//     PlcTask Outputs/GVL_iXlinker.EtherCAT_Master_EPPxxxx.Beckhoff_EPP2xxx.Beckhoff_EPP2xxxEK1122.A_0071_EPP2809_0021_0016.Channel_5.Output <-> Channel 5/Output
//     PlcTask Outputs/GVL_iXlinker.EtherCAT_Master_EPPxxxx.Beckhoff_EPP2xxx.Beckhoff_EPP2xxxEK1122.A_0071_EPP2809_0021_0016.Channel_6.Output <-> Channel 6/Output
//     PlcTask Outputs/GVL_iXlinker.EtherCAT_Master_EPPxxxx.Beckhoff_EPP2xxx.Beckhoff_EPP2xxxEK1122.A_0071_EPP2809_0021_0016.Channel_7.Output <-> Channel 7/Output
//     PlcTask Outputs/GVL_iXlinker.EtherCAT_Master_EPPxxxx.Beckhoff_EPP2xxx.Beckhoff_EPP2xxxEK1122.A_0071_EPP2809_0021_0016.Channel_8.Output <-> Channel 8/Output
//     PlcTask Outputs/GVL_iXlinker.EtherCAT_Master_EPPxxxx.Beckhoff_EPP2xxx.Beckhoff_EPP2xxxEK1122.A_0071_EPP2809_0021_0016.Channel_9.Output <-> Channel 9/Output
//     PlcTask Outputs/GVL_iXlinker.EtherCAT_Master_EPPxxxx.Beckhoff_EPP2xxx.Beckhoff_EPP2xxxEK1122.A_0071_EPP2809_0021_0016.Channel_10.Output <-> Channel 10/Output
//     PlcTask Outputs/GVL_iXlinker.EtherCAT_Master_EPPxxxx.Beckhoff_EPP2xxx.Beckhoff_EPP2xxxEK1122.A_0071_EPP2809_0021_0016.Channel_11.Output <-> Channel 11/Output
//     PlcTask Outputs/GVL_iXlinker.EtherCAT_Master_EPPxxxx.Beckhoff_EPP2xxx.Beckhoff_EPP2xxxEK1122.A_0071_EPP2809_0021_0016.Channel_12.Output <-> Channel 12/Output
//     PlcTask Outputs/GVL_iXlinker.EtherCAT_Master_EPPxxxx.Beckhoff_EPP2xxx.Beckhoff_EPP2xxxEK1122.A_0071_EPP2809_0021_0016.Channel_13.Output <-> Channel 13/Output
//     PlcTask Outputs/GVL_iXlinker.EtherCAT_Master_EPPxxxx.Beckhoff_EPP2xxx.Beckhoff_EPP2xxxEK1122.A_0071_EPP2809_0021_0016.Channel_14.Output <-> Channel 14/Output
//     PlcTask Outputs/GVL_iXlinker.EtherCAT_Master_EPPxxxx.Beckhoff_EPP2xxx.Beckhoff_EPP2xxxEK1122.A_0071_EPP2809_0021_0016.Channel_15.Output <-> Channel 15/Output
//     PlcTask Outputs/GVL_iXlinker.EtherCAT_Master_EPPxxxx.Beckhoff_EPP2xxx.Beckhoff_EPP2xxxEK1122.A_0071_EPP2809_0021_0016.Channel_16.Output <-> Channel 16/Output
//     PlcTask Inputs/GVL_iXlinker.EtherCAT_Master_EPPxxxx.Beckhoff_EPP2xxx.Beckhoff_EPP2xxxEK1122.A_0071_EPP2809_0021_0016.WcState.WcState <-> WcState/WcState
//     PlcTask Inputs/GVL_iXlinker.EtherCAT_Master_EPPxxxx.Beckhoff_EPP2xxx.Beckhoff_EPP2xxxEK1122.A_0071_EPP2809_0021_0016.InfoData.State <-> InfoData/State
//   PLC/PLC Instance <-> EtherCAT Master EPPxxxx/Beckhoff EPP2xxx/Beckhoff EPP2xxxEK1122/A_0072(EPP2809-0022-0016)
//     PlcTask Outputs/GVL_iXlinker.EtherCAT_Master_EPPxxxx.Beckhoff_EPP2xxx.Beckhoff_EPP2xxxEK1122.A_0072_EPP2809_0022_0016.Channel_1.Output <-> Channel 1/Output
//     PlcTask Outputs/GVL_iXlinker.EtherCAT_Master_EPPxxxx.Beckhoff_EPP2xxx.Beckhoff_EPP2xxxEK1122.A_0072_EPP2809_0022_0016.Channel_2.Output <-> Channel 2/Output
//     PlcTask Outputs/GVL_iXlinker.EtherCAT_Master_EPPxxxx.Beckhoff_EPP2xxx.Beckhoff_EPP2xxxEK1122.A_0072_EPP2809_0022_0016.Channel_3.Output <-> Channel 3/Output
//     PlcTask Outputs/GVL_iXlinker.EtherCAT_Master_EPPxxxx.Beckhoff_EPP2xxx.Beckhoff_EPP2xxxEK1122.A_0072_EPP2809_0022_0016.Channel_4.Output <-> Channel 4/Output
//     PlcTask Outputs/GVL_iXlinker.EtherCAT_Master_EPPxxxx.Beckhoff_EPP2xxx.Beckhoff_EPP2xxxEK1122.A_0072_EPP2809_0022_0016.Channel_5.Output <-> Channel 5/Output
//     PlcTask Outputs/GVL_iXlinker.EtherCAT_Master_EPPxxxx.Beckhoff_EPP2xxx.Beckhoff_EPP2xxxEK1122.A_0072_EPP2809_0022_0016.Channel_6.Output <-> Channel 6/Output
//     PlcTask Outputs/GVL_iXlinker.EtherCAT_Master_EPPxxxx.Beckhoff_EPP2xxx.Beckhoff_EPP2xxxEK1122.A_0072_EPP2809_0022_0016.Channel_7.Output <-> Channel 7/Output
//     PlcTask Outputs/GVL_iXlinker.EtherCAT_Master_EPPxxxx.Beckhoff_EPP2xxx.Beckhoff_EPP2xxxEK1122.A_0072_EPP2809_0022_0016.Channel_8.Output <-> Channel 8/Output
//     PlcTask Outputs/GVL_iXlinker.EtherCAT_Master_EPPxxxx.Beckhoff_EPP2xxx.Beckhoff_EPP2xxxEK1122.A_0072_EPP2809_0022_0016.Channel_9.Output <-> Channel 9/Output
//     PlcTask Outputs/GVL_iXlinker.EtherCAT_Master_EPPxxxx.Beckhoff_EPP2xxx.Beckhoff_EPP2xxxEK1122.A_0072_EPP2809_0022_0016.Channel_10.Output <-> Channel 10/Output
//     PlcTask Outputs/GVL_iXlinker.EtherCAT_Master_EPPxxxx.Beckhoff_EPP2xxx.Beckhoff_EPP2xxxEK1122.A_0072_EPP2809_0022_0016.Channel_11.Output <-> Channel 11/Output
//     PlcTask Outputs/GVL_iXlinker.EtherCAT_Master_EPPxxxx.Beckhoff_EPP2xxx.Beckhoff_EPP2xxxEK1122.A_0072_EPP2809_0022_0016.Channel_12.Output <-> Channel 12/Output
//     PlcTask Outputs/GVL_iXlinker.EtherCAT_Master_EPPxxxx.Beckhoff_EPP2xxx.Beckhoff_EPP2xxxEK1122.A_0072_EPP2809_0022_0016.Channel_13.Output <-> Channel 13/Output
//     PlcTask Outputs/GVL_iXlinker.EtherCAT_Master_EPPxxxx.Beckhoff_EPP2xxx.Beckhoff_EPP2xxxEK1122.A_0072_EPP2809_0022_0016.Channel_14.Output <-> Channel 14/Output
//     PlcTask Outputs/GVL_iXlinker.EtherCAT_Master_EPPxxxx.Beckhoff_EPP2xxx.Beckhoff_EPP2xxxEK1122.A_0072_EPP2809_0022_0016.Channel_15.Output <-> Channel 15/Output
//     PlcTask Outputs/GVL_iXlinker.EtherCAT_Master_EPPxxxx.Beckhoff_EPP2xxx.Beckhoff_EPP2xxxEK1122.A_0072_EPP2809_0022_0016.Channel_16.Output <-> Channel 16/Output
//     PlcTask Inputs/GVL_iXlinker.EtherCAT_Master_EPPxxxx.Beckhoff_EPP2xxx.Beckhoff_EPP2xxxEK1122.A_0072_EPP2809_0022_0016.WcState.WcState <-> WcState/WcState
//     PlcTask Inputs/GVL_iXlinker.EtherCAT_Master_EPPxxxx.Beckhoff_EPP2xxx.Beckhoff_EPP2xxxEK1122.A_0072_EPP2809_0022_0016.InfoData.State <-> InfoData/State
//   PLC/PLC Instance <-> EtherCAT Master EPPxxxx/Beckhoff EPP2xxx/Beckhoff EPP2xxxEK1122/A_0073(EPP2816-0004-0016)
//     PlcTask Inputs/GVL_iXlinker.EtherCAT_Master_EPPxxxx.Beckhoff_EPP2xxx.Beckhoff_EPP2xxxEK1122.A_0073_EPP2816_0004_0016.DIG_Diag_Inputs_Channel_1.Diag_Input[0] <-> DIG Diag Inputs Channel 1/Diag Input 1
//     PlcTask Inputs/GVL_iXlinker.EtherCAT_Master_EPPxxxx.Beckhoff_EPP2xxx.Beckhoff_EPP2xxxEK1122.A_0073_EPP2816_0004_0016.DIG_Diag_Inputs_Channel_1.Diag_Input[1] <-> DIG Diag Inputs Channel 1/Diag Input 2
//     PlcTask Inputs/GVL_iXlinker.EtherCAT_Master_EPPxxxx.Beckhoff_EPP2xxx.Beckhoff_EPP2xxxEK1122.A_0073_EPP2816_0004_0016.DIG_Diag_Inputs_Channel_1.Diag_Input[2] <-> DIG Diag Inputs Channel 1/Diag Input 3
//     PlcTask Inputs/GVL_iXlinker.EtherCAT_Master_EPPxxxx.Beckhoff_EPP2xxx.Beckhoff_EPP2xxxEK1122.A_0073_EPP2816_0004_0016.DIG_Diag_Inputs_Channel_1.Diag_Input[3] <-> DIG Diag Inputs Channel 1/Diag Input 4
//     PlcTask Inputs/GVL_iXlinker.EtherCAT_Master_EPPxxxx.Beckhoff_EPP2xxx.Beckhoff_EPP2xxxEK1122.A_0073_EPP2816_0004_0016.DIG_Diag_Inputs_Channel_1.Diag_Input[4] <-> DIG Diag Inputs Channel 1/Diag Input 5
//     PlcTask Inputs/GVL_iXlinker.EtherCAT_Master_EPPxxxx.Beckhoff_EPP2xxx.Beckhoff_EPP2xxxEK1122.A_0073_EPP2816_0004_0016.DIG_Diag_Inputs_Channel_1.Diag_Input[5] <-> DIG Diag Inputs Channel 1/Diag Input 6
//     PlcTask Inputs/GVL_iXlinker.EtherCAT_Master_EPPxxxx.Beckhoff_EPP2xxx.Beckhoff_EPP2xxxEK1122.A_0073_EPP2816_0004_0016.DIG_Diag_Inputs_Channel_1.Diag_Input[6] <-> DIG Diag Inputs Channel 1/Diag Input 7
//     PlcTask Inputs/GVL_iXlinker.EtherCAT_Master_EPPxxxx.Beckhoff_EPP2xxx.Beckhoff_EPP2xxxEK1122.A_0073_EPP2816_0004_0016.DIG_Diag_Inputs_Channel_1.Diag_Input[7] <-> DIG Diag Inputs Channel 1/Diag Input 8
//     PlcTask Inputs/GVL_iXlinker.EtherCAT_Master_EPPxxxx.Beckhoff_EPP2xxx.Beckhoff_EPP2xxxEK1122.A_0073_EPP2816_0004_0016.DIG_Diag_Inputs_Channel_2.Diag_Input[0] <-> DIG Diag Inputs Channel 2/Diag Input 1
//     PlcTask Inputs/GVL_iXlinker.EtherCAT_Master_EPPxxxx.Beckhoff_EPP2xxx.Beckhoff_EPP2xxxEK1122.A_0073_EPP2816_0004_0016.DIG_Diag_Inputs_Channel_2.Diag_Input[1] <-> DIG Diag Inputs Channel 2/Diag Input 2
//     PlcTask Inputs/GVL_iXlinker.EtherCAT_Master_EPPxxxx.Beckhoff_EPP2xxx.Beckhoff_EPP2xxxEK1122.A_0073_EPP2816_0004_0016.DIG_Diag_Inputs_Channel_2.Diag_Input[2] <-> DIG Diag Inputs Channel 2/Diag Input 3
//     PlcTask Inputs/GVL_iXlinker.EtherCAT_Master_EPPxxxx.Beckhoff_EPP2xxx.Beckhoff_EPP2xxxEK1122.A_0073_EPP2816_0004_0016.DIG_Diag_Inputs_Channel_2.Diag_Input[3] <-> DIG Diag Inputs Channel 2/Diag Input 4
//     PlcTask Inputs/GVL_iXlinker.EtherCAT_Master_EPPxxxx.Beckhoff_EPP2xxx.Beckhoff_EPP2xxxEK1122.A_0073_EPP2816_0004_0016.DIG_Diag_Inputs_Channel_2.Diag_Input[4] <-> DIG Diag Inputs Channel 2/Diag Input 5
//     PlcTask Inputs/GVL_iXlinker.EtherCAT_Master_EPPxxxx.Beckhoff_EPP2xxx.Beckhoff_EPP2xxxEK1122.A_0073_EPP2816_0004_0016.DIG_Diag_Inputs_Channel_2.Diag_Input[5] <-> DIG Diag Inputs Channel 2/Diag Input 6
//     PlcTask Inputs/GVL_iXlinker.EtherCAT_Master_EPPxxxx.Beckhoff_EPP2xxx.Beckhoff_EPP2xxxEK1122.A_0073_EPP2816_0004_0016.DIG_Diag_Inputs_Channel_2.Diag_Input[6] <-> DIG Diag Inputs Channel 2/Diag Input 7
//     PlcTask Inputs/GVL_iXlinker.EtherCAT_Master_EPPxxxx.Beckhoff_EPP2xxx.Beckhoff_EPP2xxxEK1122.A_0073_EPP2816_0004_0016.DIG_Diag_Inputs_Channel_2.Diag_Input[7] <-> DIG Diag Inputs Channel 2/Diag Input 8
//     PlcTask Inputs/GVL_iXlinker.EtherCAT_Master_EPPxxxx.Beckhoff_EPP2xxx.Beckhoff_EPP2xxxEK1122.A_0073_EPP2816_0004_0016.DIG_Inputs_Device.Safe_state_active <-> DIG Inputs Device/Safe state active
//     PlcTask Inputs/GVL_iXlinker.EtherCAT_Master_EPPxxxx.Beckhoff_EPP2xxx.Beckhoff_EPP2xxxEK1122.A_0073_EPP2816_0004_0016.DIG_Inputs_Device.Error_channel[0] <-> DIG Inputs Device/Error channel 1
//     PlcTask Inputs/GVL_iXlinker.EtherCAT_Master_EPPxxxx.Beckhoff_EPP2xxx.Beckhoff_EPP2xxxEK1122.A_0073_EPP2816_0004_0016.DIG_Inputs_Device.Error_channel[1] <-> DIG Inputs Device/Error channel 2
//     PlcTask Inputs/GVL_iXlinker.EtherCAT_Master_EPPxxxx.Beckhoff_EPP2xxx.Beckhoff_EPP2xxxEK1122.A_0073_EPP2816_0004_0016.DIG_Inputs_Device.Sync_error <-> DIG Inputs Device/Sync error
//     PlcTask Inputs/GVL_iXlinker.EtherCAT_Master_EPPxxxx.Beckhoff_EPP2xxx.Beckhoff_EPP2xxxEK1122.A_0073_EPP2816_0004_0016.DIG_Inputs_Device.TxPDO_Toggle <-> DIG Inputs Device/TxPDO Toggle
//     PlcTask Outputs/GVL_iXlinker.EtherCAT_Master_EPPxxxx.Beckhoff_EPP2xxx.Beckhoff_EPP2xxxEK1122.A_0073_EPP2816_0004_0016.DIG_Output_Channel_1.Output[0] <-> DIG Output Channel 1/Output 1
//     PlcTask Outputs/GVL_iXlinker.EtherCAT_Master_EPPxxxx.Beckhoff_EPP2xxx.Beckhoff_EPP2xxxEK1122.A_0073_EPP2816_0004_0016.DIG_Output_Channel_1.Output[1] <-> DIG Output Channel 1/Output 2
//     PlcTask Outputs/GVL_iXlinker.EtherCAT_Master_EPPxxxx.Beckhoff_EPP2xxx.Beckhoff_EPP2xxxEK1122.A_0073_EPP2816_0004_0016.DIG_Output_Channel_1.Output[2] <-> DIG Output Channel 1/Output 3
//     PlcTask Outputs/GVL_iXlinker.EtherCAT_Master_EPPxxxx.Beckhoff_EPP2xxx.Beckhoff_EPP2xxxEK1122.A_0073_EPP2816_0004_0016.DIG_Output_Channel_1.Output[3] <-> DIG Output Channel 1/Output 4
//     PlcTask Outputs/GVL_iXlinker.EtherCAT_Master_EPPxxxx.Beckhoff_EPP2xxx.Beckhoff_EPP2xxxEK1122.A_0073_EPP2816_0004_0016.DIG_Output_Channel_1.Output[4] <-> DIG Output Channel 1/Output 5
//     PlcTask Outputs/GVL_iXlinker.EtherCAT_Master_EPPxxxx.Beckhoff_EPP2xxx.Beckhoff_EPP2xxxEK1122.A_0073_EPP2816_0004_0016.DIG_Output_Channel_1.Output[5] <-> DIG Output Channel 1/Output 6
//     PlcTask Outputs/GVL_iXlinker.EtherCAT_Master_EPPxxxx.Beckhoff_EPP2xxx.Beckhoff_EPP2xxxEK1122.A_0073_EPP2816_0004_0016.DIG_Output_Channel_1.Output[6] <-> DIG Output Channel 1/Output 7
//     PlcTask Outputs/GVL_iXlinker.EtherCAT_Master_EPPxxxx.Beckhoff_EPP2xxx.Beckhoff_EPP2xxxEK1122.A_0073_EPP2816_0004_0016.DIG_Output_Channel_1.Output[7] <-> DIG Output Channel 1/Output 8
//     PlcTask Outputs/GVL_iXlinker.EtherCAT_Master_EPPxxxx.Beckhoff_EPP2xxx.Beckhoff_EPP2xxxEK1122.A_0073_EPP2816_0004_0016.DIG_Output_Channel_2.Output[0] <-> DIG Output Channel 2/Output 1
//     PlcTask Outputs/GVL_iXlinker.EtherCAT_Master_EPPxxxx.Beckhoff_EPP2xxx.Beckhoff_EPP2xxxEK1122.A_0073_EPP2816_0004_0016.DIG_Output_Channel_2.Output[1] <-> DIG Output Channel 2/Output 2
//     PlcTask Outputs/GVL_iXlinker.EtherCAT_Master_EPPxxxx.Beckhoff_EPP2xxx.Beckhoff_EPP2xxxEK1122.A_0073_EPP2816_0004_0016.DIG_Output_Channel_2.Output[2] <-> DIG Output Channel 2/Output 3
//     PlcTask Outputs/GVL_iXlinker.EtherCAT_Master_EPPxxxx.Beckhoff_EPP2xxx.Beckhoff_EPP2xxxEK1122.A_0073_EPP2816_0004_0016.DIG_Output_Channel_2.Output[3] <-> DIG Output Channel 2/Output 4
//     PlcTask Outputs/GVL_iXlinker.EtherCAT_Master_EPPxxxx.Beckhoff_EPP2xxx.Beckhoff_EPP2xxxEK1122.A_0073_EPP2816_0004_0016.DIG_Output_Channel_2.Output[4] <-> DIG Output Channel 2/Output 5
//     PlcTask Outputs/GVL_iXlinker.EtherCAT_Master_EPPxxxx.Beckhoff_EPP2xxx.Beckhoff_EPP2xxxEK1122.A_0073_EPP2816_0004_0016.DIG_Output_Channel_2.Output[5] <-> DIG Output Channel 2/Output 6
//     PlcTask Outputs/GVL_iXlinker.EtherCAT_Master_EPPxxxx.Beckhoff_EPP2xxx.Beckhoff_EPP2xxxEK1122.A_0073_EPP2816_0004_0016.DIG_Output_Channel_2.Output[6] <-> DIG Output Channel 2/Output 7
//     PlcTask Outputs/GVL_iXlinker.EtherCAT_Master_EPPxxxx.Beckhoff_EPP2xxx.Beckhoff_EPP2xxxEK1122.A_0073_EPP2816_0004_0016.DIG_Output_Channel_2.Output[7] <-> DIG Output Channel 2/Output 8
//     PlcTask Outputs/GVL_iXlinker.EtherCAT_Master_EPPxxxx.Beckhoff_EPP2xxx.Beckhoff_EPP2xxxEK1122.A_0073_EPP2816_0004_0016.DIG_Outputs_Device.Set_safe_state <-> DIG Outputs Device/Set safe state
//     PlcTask Outputs/GVL_iXlinker.EtherCAT_Master_EPPxxxx.Beckhoff_EPP2xxx.Beckhoff_EPP2xxxEK1122.A_0073_EPP2816_0004_0016.DIG_Outputs_Device.Reset_outputs <-> DIG Outputs Device/Reset outputs
//     PlcTask Inputs/GVL_iXlinker.EtherCAT_Master_EPPxxxx.Beckhoff_EPP2xxx.Beckhoff_EPP2xxxEK1122.A_0073_EPP2816_0004_0016.WcState.WcState <-> WcState/WcState
//     PlcTask Inputs/GVL_iXlinker.EtherCAT_Master_EPPxxxx.Beckhoff_EPP2xxx.Beckhoff_EPP2xxxEK1122.A_0073_EPP2816_0004_0016.WcState.InputToggle <-> WcState/InputToggle
//     PlcTask Inputs/GVL_iXlinker.EtherCAT_Master_EPPxxxx.Beckhoff_EPP2xxx.Beckhoff_EPP2xxxEK1122.A_0073_EPP2816_0004_0016.InfoData.AdsAddr <-> InfoData/AdsAddr
//     PlcTask Inputs/GVL_iXlinker.EtherCAT_Master_EPPxxxx.Beckhoff_EPP2xxx.Beckhoff_EPP2xxxEK1122.A_0073_EPP2816_0004_0016.InfoData.State <-> InfoData/State
//   PLC/PLC Instance <-> EtherCAT Master EPPxxxx/Beckhoff EPP2xxx/Beckhoff EPP2xxxEK1122/A_0074(EPP2816-0004-0017)
//     PlcTask Inputs/GVL_iXlinker.EtherCAT_Master_EPPxxxx.Beckhoff_EPP2xxx.Beckhoff_EPP2xxxEK1122.A_0074_EPP2816_0004_0017.DIG_Diag_Inputs_Channel_1.Diag_Input[0] <-> DIG Diag Inputs Channel 1/Diag Input 1
//     PlcTask Inputs/GVL_iXlinker.EtherCAT_Master_EPPxxxx.Beckhoff_EPP2xxx.Beckhoff_EPP2xxxEK1122.A_0074_EPP2816_0004_0017.DIG_Diag_Inputs_Channel_1.Diag_Input[1] <-> DIG Diag Inputs Channel 1/Diag Input 2
//     PlcTask Inputs/GVL_iXlinker.EtherCAT_Master_EPPxxxx.Beckhoff_EPP2xxx.Beckhoff_EPP2xxxEK1122.A_0074_EPP2816_0004_0017.DIG_Diag_Inputs_Channel_1.Diag_Input[2] <-> DIG Diag Inputs Channel 1/Diag Input 3
//     PlcTask Inputs/GVL_iXlinker.EtherCAT_Master_EPPxxxx.Beckhoff_EPP2xxx.Beckhoff_EPP2xxxEK1122.A_0074_EPP2816_0004_0017.DIG_Diag_Inputs_Channel_1.Diag_Input[3] <-> DIG Diag Inputs Channel 1/Diag Input 4
//     PlcTask Inputs/GVL_iXlinker.EtherCAT_Master_EPPxxxx.Beckhoff_EPP2xxx.Beckhoff_EPP2xxxEK1122.A_0074_EPP2816_0004_0017.DIG_Diag_Inputs_Channel_1.Diag_Input[4] <-> DIG Diag Inputs Channel 1/Diag Input 5
//     PlcTask Inputs/GVL_iXlinker.EtherCAT_Master_EPPxxxx.Beckhoff_EPP2xxx.Beckhoff_EPP2xxxEK1122.A_0074_EPP2816_0004_0017.DIG_Diag_Inputs_Channel_1.Diag_Input[5] <-> DIG Diag Inputs Channel 1/Diag Input 6
//     PlcTask Inputs/GVL_iXlinker.EtherCAT_Master_EPPxxxx.Beckhoff_EPP2xxx.Beckhoff_EPP2xxxEK1122.A_0074_EPP2816_0004_0017.DIG_Diag_Inputs_Channel_1.Diag_Input[6] <-> DIG Diag Inputs Channel 1/Diag Input 7
//     PlcTask Inputs/GVL_iXlinker.EtherCAT_Master_EPPxxxx.Beckhoff_EPP2xxx.Beckhoff_EPP2xxxEK1122.A_0074_EPP2816_0004_0017.DIG_Diag_Inputs_Channel_1.Diag_Input[7] <-> DIG Diag Inputs Channel 1/Diag Input 8
//     PlcTask Inputs/GVL_iXlinker.EtherCAT_Master_EPPxxxx.Beckhoff_EPP2xxx.Beckhoff_EPP2xxxEK1122.A_0074_EPP2816_0004_0017.DIG_Diag_Inputs_Channel_2.Diag_Input[0] <-> DIG Diag Inputs Channel 2/Diag Input 1
//     PlcTask Inputs/GVL_iXlinker.EtherCAT_Master_EPPxxxx.Beckhoff_EPP2xxx.Beckhoff_EPP2xxxEK1122.A_0074_EPP2816_0004_0017.DIG_Diag_Inputs_Channel_2.Diag_Input[1] <-> DIG Diag Inputs Channel 2/Diag Input 2
//     PlcTask Inputs/GVL_iXlinker.EtherCAT_Master_EPPxxxx.Beckhoff_EPP2xxx.Beckhoff_EPP2xxxEK1122.A_0074_EPP2816_0004_0017.DIG_Diag_Inputs_Channel_2.Diag_Input[2] <-> DIG Diag Inputs Channel 2/Diag Input 3
//     PlcTask Inputs/GVL_iXlinker.EtherCAT_Master_EPPxxxx.Beckhoff_EPP2xxx.Beckhoff_EPP2xxxEK1122.A_0074_EPP2816_0004_0017.DIG_Diag_Inputs_Channel_2.Diag_Input[3] <-> DIG Diag Inputs Channel 2/Diag Input 4
//     PlcTask Inputs/GVL_iXlinker.EtherCAT_Master_EPPxxxx.Beckhoff_EPP2xxx.Beckhoff_EPP2xxxEK1122.A_0074_EPP2816_0004_0017.DIG_Diag_Inputs_Channel_2.Diag_Input[4] <-> DIG Diag Inputs Channel 2/Diag Input 5
//     PlcTask Inputs/GVL_iXlinker.EtherCAT_Master_EPPxxxx.Beckhoff_EPP2xxx.Beckhoff_EPP2xxxEK1122.A_0074_EPP2816_0004_0017.DIG_Diag_Inputs_Channel_2.Diag_Input[5] <-> DIG Diag Inputs Channel 2/Diag Input 6
//     PlcTask Inputs/GVL_iXlinker.EtherCAT_Master_EPPxxxx.Beckhoff_EPP2xxx.Beckhoff_EPP2xxxEK1122.A_0074_EPP2816_0004_0017.DIG_Diag_Inputs_Channel_2.Diag_Input[6] <-> DIG Diag Inputs Channel 2/Diag Input 7
//     PlcTask Inputs/GVL_iXlinker.EtherCAT_Master_EPPxxxx.Beckhoff_EPP2xxx.Beckhoff_EPP2xxxEK1122.A_0074_EPP2816_0004_0017.DIG_Diag_Inputs_Channel_2.Diag_Input[7] <-> DIG Diag Inputs Channel 2/Diag Input 8
//     PlcTask Inputs/GVL_iXlinker.EtherCAT_Master_EPPxxxx.Beckhoff_EPP2xxx.Beckhoff_EPP2xxxEK1122.A_0074_EPP2816_0004_0017.DIG_Inputs_Device.Safe_state_active <-> DIG Inputs Device/Safe state active
//     PlcTask Inputs/GVL_iXlinker.EtherCAT_Master_EPPxxxx.Beckhoff_EPP2xxx.Beckhoff_EPP2xxxEK1122.A_0074_EPP2816_0004_0017.DIG_Inputs_Device.Error_channel[0] <-> DIG Inputs Device/Error channel 1
//     PlcTask Inputs/GVL_iXlinker.EtherCAT_Master_EPPxxxx.Beckhoff_EPP2xxx.Beckhoff_EPP2xxxEK1122.A_0074_EPP2816_0004_0017.DIG_Inputs_Device.Error_channel[1] <-> DIG Inputs Device/Error channel 2
//     PlcTask Inputs/GVL_iXlinker.EtherCAT_Master_EPPxxxx.Beckhoff_EPP2xxx.Beckhoff_EPP2xxxEK1122.A_0074_EPP2816_0004_0017.DIG_Inputs_Device.Sync_error <-> DIG Inputs Device/Sync error
//     PlcTask Inputs/GVL_iXlinker.EtherCAT_Master_EPPxxxx.Beckhoff_EPP2xxx.Beckhoff_EPP2xxxEK1122.A_0074_EPP2816_0004_0017.DIG_Inputs_Device.TxPDO_Toggle <-> DIG Inputs Device/TxPDO Toggle
//     PlcTask Outputs/GVL_iXlinker.EtherCAT_Master_EPPxxxx.Beckhoff_EPP2xxx.Beckhoff_EPP2xxxEK1122.A_0074_EPP2816_0004_0017.DIG_Output_Channel_1.Output[0] <-> DIG Output Channel 1/Output 1
//     PlcTask Outputs/GVL_iXlinker.EtherCAT_Master_EPPxxxx.Beckhoff_EPP2xxx.Beckhoff_EPP2xxxEK1122.A_0074_EPP2816_0004_0017.DIG_Output_Channel_1.Output[1] <-> DIG Output Channel 1/Output 2
//     PlcTask Outputs/GVL_iXlinker.EtherCAT_Master_EPPxxxx.Beckhoff_EPP2xxx.Beckhoff_EPP2xxxEK1122.A_0074_EPP2816_0004_0017.DIG_Output_Channel_1.Output[2] <-> DIG Output Channel 1/Output 3
//     PlcTask Outputs/GVL_iXlinker.EtherCAT_Master_EPPxxxx.Beckhoff_EPP2xxx.Beckhoff_EPP2xxxEK1122.A_0074_EPP2816_0004_0017.DIG_Output_Channel_1.Output[3] <-> DIG Output Channel 1/Output 4
//     PlcTask Outputs/GVL_iXlinker.EtherCAT_Master_EPPxxxx.Beckhoff_EPP2xxx.Beckhoff_EPP2xxxEK1122.A_0074_EPP2816_0004_0017.DIG_Output_Channel_1.Output[4] <-> DIG Output Channel 1/Output 5
//     PlcTask Outputs/GVL_iXlinker.EtherCAT_Master_EPPxxxx.Beckhoff_EPP2xxx.Beckhoff_EPP2xxxEK1122.A_0074_EPP2816_0004_0017.DIG_Output_Channel_1.Output[5] <-> DIG Output Channel 1/Output 6
//     PlcTask Outputs/GVL_iXlinker.EtherCAT_Master_EPPxxxx.Beckhoff_EPP2xxx.Beckhoff_EPP2xxxEK1122.A_0074_EPP2816_0004_0017.DIG_Output_Channel_1.Output[6] <-> DIG Output Channel 1/Output 7
//     PlcTask Outputs/GVL_iXlinker.EtherCAT_Master_EPPxxxx.Beckhoff_EPP2xxx.Beckhoff_EPP2xxxEK1122.A_0074_EPP2816_0004_0017.DIG_Output_Channel_1.Output[7] <-> DIG Output Channel 1/Output 8
//     PlcTask Outputs/GVL_iXlinker.EtherCAT_Master_EPPxxxx.Beckhoff_EPP2xxx.Beckhoff_EPP2xxxEK1122.A_0074_EPP2816_0004_0017.DIG_Output_Channel_2.Output[0] <-> DIG Output Channel 2/Output 1
//     PlcTask Outputs/GVL_iXlinker.EtherCAT_Master_EPPxxxx.Beckhoff_EPP2xxx.Beckhoff_EPP2xxxEK1122.A_0074_EPP2816_0004_0017.DIG_Output_Channel_2.Output[1] <-> DIG Output Channel 2/Output 2
//     PlcTask Outputs/GVL_iXlinker.EtherCAT_Master_EPPxxxx.Beckhoff_EPP2xxx.Beckhoff_EPP2xxxEK1122.A_0074_EPP2816_0004_0017.DIG_Output_Channel_2.Output[2] <-> DIG Output Channel 2/Output 3
//     PlcTask Outputs/GVL_iXlinker.EtherCAT_Master_EPPxxxx.Beckhoff_EPP2xxx.Beckhoff_EPP2xxxEK1122.A_0074_EPP2816_0004_0017.DIG_Output_Channel_2.Output[3] <-> DIG Output Channel 2/Output 4
//     PlcTask Outputs/GVL_iXlinker.EtherCAT_Master_EPPxxxx.Beckhoff_EPP2xxx.Beckhoff_EPP2xxxEK1122.A_0074_EPP2816_0004_0017.DIG_Output_Channel_2.Output[4] <-> DIG Output Channel 2/Output 5
//     PlcTask Outputs/GVL_iXlinker.EtherCAT_Master_EPPxxxx.Beckhoff_EPP2xxx.Beckhoff_EPP2xxxEK1122.A_0074_EPP2816_0004_0017.DIG_Output_Channel_2.Output[5] <-> DIG Output Channel 2/Output 6
//     PlcTask Outputs/GVL_iXlinker.EtherCAT_Master_EPPxxxx.Beckhoff_EPP2xxx.Beckhoff_EPP2xxxEK1122.A_0074_EPP2816_0004_0017.DIG_Output_Channel_2.Output[6] <-> DIG Output Channel 2/Output 7
//     PlcTask Outputs/GVL_iXlinker.EtherCAT_Master_EPPxxxx.Beckhoff_EPP2xxx.Beckhoff_EPP2xxxEK1122.A_0074_EPP2816_0004_0017.DIG_Output_Channel_2.Output[7] <-> DIG Output Channel 2/Output 8
//     PlcTask Outputs/GVL_iXlinker.EtherCAT_Master_EPPxxxx.Beckhoff_EPP2xxx.Beckhoff_EPP2xxxEK1122.A_0074_EPP2816_0004_0017.DIG_Outputs_Device.Set_safe_state <-> DIG Outputs Device/Set safe state
//     PlcTask Outputs/GVL_iXlinker.EtherCAT_Master_EPPxxxx.Beckhoff_EPP2xxx.Beckhoff_EPP2xxxEK1122.A_0074_EPP2816_0004_0017.DIG_Outputs_Device.Reset_outputs <-> DIG Outputs Device/Reset outputs
//     PlcTask Inputs/GVL_iXlinker.EtherCAT_Master_EPPxxxx.Beckhoff_EPP2xxx.Beckhoff_EPP2xxxEK1122.A_0074_EPP2816_0004_0017.WcState.WcState <-> WcState/WcState
//     PlcTask Inputs/GVL_iXlinker.EtherCAT_Master_EPPxxxx.Beckhoff_EPP2xxx.Beckhoff_EPP2xxxEK1122.A_0074_EPP2816_0004_0017.WcState.InputToggle <-> WcState/InputToggle
//     PlcTask Inputs/GVL_iXlinker.EtherCAT_Master_EPPxxxx.Beckhoff_EPP2xxx.Beckhoff_EPP2xxxEK1122.A_0074_EPP2816_0004_0017.InfoData.AdsAddr <-> InfoData/AdsAddr
//     PlcTask Inputs/GVL_iXlinker.EtherCAT_Master_EPPxxxx.Beckhoff_EPP2xxx.Beckhoff_EPP2xxxEK1122.A_0074_EPP2816_0004_0017.InfoData.State <-> InfoData/State
//   PLC/PLC Instance <-> EtherCAT Master EPPxxxx/Beckhoff EPP2xxx/Beckhoff EPP2xxxEK1122/A_0075(EPP2816-0008-0016)
//     PlcTask Inputs/GVL_iXlinker.EtherCAT_Master_EPPxxxx.Beckhoff_EPP2xxx.Beckhoff_EPP2xxxEK1122.A_0075_EPP2816_0008_0016.DIG_Diag_Inputs_Channel_1.Diag_Input[0] <-> DIG Diag Inputs  Channel 1/Diag Input 1
//     PlcTask Inputs/GVL_iXlinker.EtherCAT_Master_EPPxxxx.Beckhoff_EPP2xxx.Beckhoff_EPP2xxxEK1122.A_0075_EPP2816_0008_0016.DIG_Diag_Inputs_Channel_1.Diag_Input[1] <-> DIG Diag Inputs  Channel 1/Diag Input 2
//     PlcTask Inputs/GVL_iXlinker.EtherCAT_Master_EPPxxxx.Beckhoff_EPP2xxx.Beckhoff_EPP2xxxEK1122.A_0075_EPP2816_0008_0016.DIG_Diag_Inputs_Channel_1.Diag_Input[2] <-> DIG Diag Inputs  Channel 1/Diag Input 3
//     PlcTask Inputs/GVL_iXlinker.EtherCAT_Master_EPPxxxx.Beckhoff_EPP2xxx.Beckhoff_EPP2xxxEK1122.A_0075_EPP2816_0008_0016.DIG_Diag_Inputs_Channel_1.Diag_Input[3] <-> DIG Diag Inputs  Channel 1/Diag Input 4
//     PlcTask Inputs/GVL_iXlinker.EtherCAT_Master_EPPxxxx.Beckhoff_EPP2xxx.Beckhoff_EPP2xxxEK1122.A_0075_EPP2816_0008_0016.DIG_Diag_Inputs_Channel_1.Diag_Input[4] <-> DIG Diag Inputs  Channel 1/Diag Input 5
//     PlcTask Inputs/GVL_iXlinker.EtherCAT_Master_EPPxxxx.Beckhoff_EPP2xxx.Beckhoff_EPP2xxxEK1122.A_0075_EPP2816_0008_0016.DIG_Diag_Inputs_Channel_1.Diag_Input[5] <-> DIG Diag Inputs  Channel 1/Diag Input 6
//     PlcTask Inputs/GVL_iXlinker.EtherCAT_Master_EPPxxxx.Beckhoff_EPP2xxx.Beckhoff_EPP2xxxEK1122.A_0075_EPP2816_0008_0016.DIG_Diag_Inputs_Channel_1.Diag_Input[6] <-> DIG Diag Inputs  Channel 1/Diag Input 7
//     PlcTask Inputs/GVL_iXlinker.EtherCAT_Master_EPPxxxx.Beckhoff_EPP2xxx.Beckhoff_EPP2xxxEK1122.A_0075_EPP2816_0008_0016.DIG_Diag_Inputs_Channel_1.Diag_Input[7] <-> DIG Diag Inputs  Channel 1/Diag Input 8
//     PlcTask Inputs/GVL_iXlinker.EtherCAT_Master_EPPxxxx.Beckhoff_EPP2xxx.Beckhoff_EPP2xxxEK1122.A_0075_EPP2816_0008_0016.DIG_Diag_Inputs_Channel_2.Diag_Input[0] <-> DIG Diag Inputs  Channel 2/Diag Input 1
//     PlcTask Inputs/GVL_iXlinker.EtherCAT_Master_EPPxxxx.Beckhoff_EPP2xxx.Beckhoff_EPP2xxxEK1122.A_0075_EPP2816_0008_0016.DIG_Diag_Inputs_Channel_2.Diag_Input[1] <-> DIG Diag Inputs  Channel 2/Diag Input 2
//     PlcTask Inputs/GVL_iXlinker.EtherCAT_Master_EPPxxxx.Beckhoff_EPP2xxx.Beckhoff_EPP2xxxEK1122.A_0075_EPP2816_0008_0016.DIG_Diag_Inputs_Channel_2.Diag_Input[2] <-> DIG Diag Inputs  Channel 2/Diag Input 3
//     PlcTask Inputs/GVL_iXlinker.EtherCAT_Master_EPPxxxx.Beckhoff_EPP2xxx.Beckhoff_EPP2xxxEK1122.A_0075_EPP2816_0008_0016.DIG_Diag_Inputs_Channel_2.Diag_Input[3] <-> DIG Diag Inputs  Channel 2/Diag Input 4
//     PlcTask Inputs/GVL_iXlinker.EtherCAT_Master_EPPxxxx.Beckhoff_EPP2xxx.Beckhoff_EPP2xxxEK1122.A_0075_EPP2816_0008_0016.DIG_Diag_Inputs_Channel_2.Diag_Input[4] <-> DIG Diag Inputs  Channel 2/Diag Input 5
//     PlcTask Inputs/GVL_iXlinker.EtherCAT_Master_EPPxxxx.Beckhoff_EPP2xxx.Beckhoff_EPP2xxxEK1122.A_0075_EPP2816_0008_0016.DIG_Diag_Inputs_Channel_2.Diag_Input[5] <-> DIG Diag Inputs  Channel 2/Diag Input 6
//     PlcTask Inputs/GVL_iXlinker.EtherCAT_Master_EPPxxxx.Beckhoff_EPP2xxx.Beckhoff_EPP2xxxEK1122.A_0075_EPP2816_0008_0016.DIG_Diag_Inputs_Channel_2.Diag_Input[6] <-> DIG Diag Inputs  Channel 2/Diag Input 7
//     PlcTask Inputs/GVL_iXlinker.EtherCAT_Master_EPPxxxx.Beckhoff_EPP2xxx.Beckhoff_EPP2xxxEK1122.A_0075_EPP2816_0008_0016.DIG_Diag_Inputs_Channel_2.Diag_Input[7] <-> DIG Diag Inputs  Channel 2/Diag Input 8
//     PlcTask Inputs/GVL_iXlinker.EtherCAT_Master_EPPxxxx.Beckhoff_EPP2xxx.Beckhoff_EPP2xxxEK1122.A_0075_EPP2816_0008_0016.DIG_Inputs_Device.Safe_state_active <-> DIG Inputs Device/Safe state active
//     PlcTask Inputs/GVL_iXlinker.EtherCAT_Master_EPPxxxx.Beckhoff_EPP2xxx.Beckhoff_EPP2xxxEK1122.A_0075_EPP2816_0008_0016.DIG_Inputs_Device.Error_channel[0] <-> DIG Inputs Device/Error channel 1
//     PlcTask Inputs/GVL_iXlinker.EtherCAT_Master_EPPxxxx.Beckhoff_EPP2xxx.Beckhoff_EPP2xxxEK1122.A_0075_EPP2816_0008_0016.DIG_Inputs_Device.Error_channel[1] <-> DIG Inputs Device/Error channel 2
//     PlcTask Inputs/GVL_iXlinker.EtherCAT_Master_EPPxxxx.Beckhoff_EPP2xxx.Beckhoff_EPP2xxxEK1122.A_0075_EPP2816_0008_0016.DIG_Inputs_Device.Sync_error <-> DIG Inputs Device/Sync error
//     PlcTask Inputs/GVL_iXlinker.EtherCAT_Master_EPPxxxx.Beckhoff_EPP2xxx.Beckhoff_EPP2xxxEK1122.A_0075_EPP2816_0008_0016.DIG_Inputs_Device.TxPDO_Toggle <-> DIG Inputs Device/TxPDO Toggle
//     PlcTask Outputs/GVL_iXlinker.EtherCAT_Master_EPPxxxx.Beckhoff_EPP2xxx.Beckhoff_EPP2xxxEK1122.A_0075_EPP2816_0008_0016.DIG_Outputs_Channel_1.Output[0] <-> DIG Outputs Channel 1/Output 1
//     PlcTask Outputs/GVL_iXlinker.EtherCAT_Master_EPPxxxx.Beckhoff_EPP2xxx.Beckhoff_EPP2xxxEK1122.A_0075_EPP2816_0008_0016.DIG_Outputs_Channel_1.Output[1] <-> DIG Outputs Channel 1/Output 2
//     PlcTask Outputs/GVL_iXlinker.EtherCAT_Master_EPPxxxx.Beckhoff_EPP2xxx.Beckhoff_EPP2xxxEK1122.A_0075_EPP2816_0008_0016.DIG_Outputs_Channel_1.Output[2] <-> DIG Outputs Channel 1/Output 3
//     PlcTask Outputs/GVL_iXlinker.EtherCAT_Master_EPPxxxx.Beckhoff_EPP2xxx.Beckhoff_EPP2xxxEK1122.A_0075_EPP2816_0008_0016.DIG_Outputs_Channel_1.Output[3] <-> DIG Outputs Channel 1/Output 4
//     PlcTask Outputs/GVL_iXlinker.EtherCAT_Master_EPPxxxx.Beckhoff_EPP2xxx.Beckhoff_EPP2xxxEK1122.A_0075_EPP2816_0008_0016.DIG_Outputs_Channel_1.Output[4] <-> DIG Outputs Channel 1/Output 5
//     PlcTask Outputs/GVL_iXlinker.EtherCAT_Master_EPPxxxx.Beckhoff_EPP2xxx.Beckhoff_EPP2xxxEK1122.A_0075_EPP2816_0008_0016.DIG_Outputs_Channel_1.Output[5] <-> DIG Outputs Channel 1/Output 6
//     PlcTask Outputs/GVL_iXlinker.EtherCAT_Master_EPPxxxx.Beckhoff_EPP2xxx.Beckhoff_EPP2xxxEK1122.A_0075_EPP2816_0008_0016.DIG_Outputs_Channel_1.Output[6] <-> DIG Outputs Channel 1/Output 7
//     PlcTask Outputs/GVL_iXlinker.EtherCAT_Master_EPPxxxx.Beckhoff_EPP2xxx.Beckhoff_EPP2xxxEK1122.A_0075_EPP2816_0008_0016.DIG_Outputs_Channel_1.Output[7] <-> DIG Outputs Channel 1/Output 8
//     PlcTask Outputs/GVL_iXlinker.EtherCAT_Master_EPPxxxx.Beckhoff_EPP2xxx.Beckhoff_EPP2xxxEK1122.A_0075_EPP2816_0008_0016.DIG_Outputs_Channel_2.Output[0] <-> DIG Outputs Channel 2/Output 1
//     PlcTask Outputs/GVL_iXlinker.EtherCAT_Master_EPPxxxx.Beckhoff_EPP2xxx.Beckhoff_EPP2xxxEK1122.A_0075_EPP2816_0008_0016.DIG_Outputs_Channel_2.Output[1] <-> DIG Outputs Channel 2/Output 2
//     PlcTask Outputs/GVL_iXlinker.EtherCAT_Master_EPPxxxx.Beckhoff_EPP2xxx.Beckhoff_EPP2xxxEK1122.A_0075_EPP2816_0008_0016.DIG_Outputs_Channel_2.Output[2] <-> DIG Outputs Channel 2/Output 3
//     PlcTask Outputs/GVL_iXlinker.EtherCAT_Master_EPPxxxx.Beckhoff_EPP2xxx.Beckhoff_EPP2xxxEK1122.A_0075_EPP2816_0008_0016.DIG_Outputs_Channel_2.Output[3] <-> DIG Outputs Channel 2/Output 4
//     PlcTask Outputs/GVL_iXlinker.EtherCAT_Master_EPPxxxx.Beckhoff_EPP2xxx.Beckhoff_EPP2xxxEK1122.A_0075_EPP2816_0008_0016.DIG_Outputs_Channel_2.Output[4] <-> DIG Outputs Channel 2/Output 5
//     PlcTask Outputs/GVL_iXlinker.EtherCAT_Master_EPPxxxx.Beckhoff_EPP2xxx.Beckhoff_EPP2xxxEK1122.A_0075_EPP2816_0008_0016.DIG_Outputs_Channel_2.Output[5] <-> DIG Outputs Channel 2/Output 6
//     PlcTask Outputs/GVL_iXlinker.EtherCAT_Master_EPPxxxx.Beckhoff_EPP2xxx.Beckhoff_EPP2xxxEK1122.A_0075_EPP2816_0008_0016.DIG_Outputs_Channel_2.Output[6] <-> DIG Outputs Channel 2/Output 7
//     PlcTask Outputs/GVL_iXlinker.EtherCAT_Master_EPPxxxx.Beckhoff_EPP2xxx.Beckhoff_EPP2xxxEK1122.A_0075_EPP2816_0008_0016.DIG_Outputs_Channel_2.Output[7] <-> DIG Outputs Channel 2/Output 8
//     PlcTask Outputs/GVL_iXlinker.EtherCAT_Master_EPPxxxx.Beckhoff_EPP2xxx.Beckhoff_EPP2xxxEK1122.A_0075_EPP2816_0008_0016.DIG_Outputs_Device.Set_safe_state <-> DIG Outputs Device/Set safe state
//     PlcTask Outputs/GVL_iXlinker.EtherCAT_Master_EPPxxxx.Beckhoff_EPP2xxx.Beckhoff_EPP2xxxEK1122.A_0075_EPP2816_0008_0016.DIG_Outputs_Device.Reset_outputs <-> DIG Outputs Device/Reset outputs
//     PlcTask Inputs/GVL_iXlinker.EtherCAT_Master_EPPxxxx.Beckhoff_EPP2xxx.Beckhoff_EPP2xxxEK1122.A_0075_EPP2816_0008_0016.WcState.WcState <-> WcState/WcState
//     PlcTask Inputs/GVL_iXlinker.EtherCAT_Master_EPPxxxx.Beckhoff_EPP2xxx.Beckhoff_EPP2xxxEK1122.A_0075_EPP2816_0008_0016.WcState.InputToggle <-> WcState/InputToggle
//     PlcTask Inputs/GVL_iXlinker.EtherCAT_Master_EPPxxxx.Beckhoff_EPP2xxx.Beckhoff_EPP2xxxEK1122.A_0075_EPP2816_0008_0016.InfoData.AdsAddr <-> InfoData/AdsAddr
//     PlcTask Inputs/GVL_iXlinker.EtherCAT_Master_EPPxxxx.Beckhoff_EPP2xxx.Beckhoff_EPP2xxxEK1122.A_0075_EPP2816_0008_0016.InfoData.State <-> InfoData/State
//   PLC/PLC Instance <-> EtherCAT Master EPPxxxx/Beckhoff EPP2xxx/Beckhoff EPP2xxxEK1122/A_0076(EPP2816-0008-0017)
//     PlcTask Inputs/GVL_iXlinker.EtherCAT_Master_EPPxxxx.Beckhoff_EPP2xxx.Beckhoff_EPP2xxxEK1122.A_0076_EPP2816_0008_0017.DIG_Diag_Inputs_Channel_1.Diag_Input[0] <-> DIG Diag Inputs  Channel 1/Diag Input 1
//     PlcTask Inputs/GVL_iXlinker.EtherCAT_Master_EPPxxxx.Beckhoff_EPP2xxx.Beckhoff_EPP2xxxEK1122.A_0076_EPP2816_0008_0017.DIG_Diag_Inputs_Channel_1.Diag_Input[1] <-> DIG Diag Inputs  Channel 1/Diag Input 2
//     PlcTask Inputs/GVL_iXlinker.EtherCAT_Master_EPPxxxx.Beckhoff_EPP2xxx.Beckhoff_EPP2xxxEK1122.A_0076_EPP2816_0008_0017.DIG_Diag_Inputs_Channel_1.Diag_Input[2] <-> DIG Diag Inputs  Channel 1/Diag Input 3
//     PlcTask Inputs/GVL_iXlinker.EtherCAT_Master_EPPxxxx.Beckhoff_EPP2xxx.Beckhoff_EPP2xxxEK1122.A_0076_EPP2816_0008_0017.DIG_Diag_Inputs_Channel_1.Diag_Input[3] <-> DIG Diag Inputs  Channel 1/Diag Input 4
//     PlcTask Inputs/GVL_iXlinker.EtherCAT_Master_EPPxxxx.Beckhoff_EPP2xxx.Beckhoff_EPP2xxxEK1122.A_0076_EPP2816_0008_0017.DIG_Diag_Inputs_Channel_1.Diag_Input[4] <-> DIG Diag Inputs  Channel 1/Diag Input 5
//     PlcTask Inputs/GVL_iXlinker.EtherCAT_Master_EPPxxxx.Beckhoff_EPP2xxx.Beckhoff_EPP2xxxEK1122.A_0076_EPP2816_0008_0017.DIG_Diag_Inputs_Channel_1.Diag_Input[5] <-> DIG Diag Inputs  Channel 1/Diag Input 6
//     PlcTask Inputs/GVL_iXlinker.EtherCAT_Master_EPPxxxx.Beckhoff_EPP2xxx.Beckhoff_EPP2xxxEK1122.A_0076_EPP2816_0008_0017.DIG_Diag_Inputs_Channel_1.Diag_Input[6] <-> DIG Diag Inputs  Channel 1/Diag Input 7
//     PlcTask Inputs/GVL_iXlinker.EtherCAT_Master_EPPxxxx.Beckhoff_EPP2xxx.Beckhoff_EPP2xxxEK1122.A_0076_EPP2816_0008_0017.DIG_Diag_Inputs_Channel_1.Diag_Input[7] <-> DIG Diag Inputs  Channel 1/Diag Input 8
//     PlcTask Inputs/GVL_iXlinker.EtherCAT_Master_EPPxxxx.Beckhoff_EPP2xxx.Beckhoff_EPP2xxxEK1122.A_0076_EPP2816_0008_0017.DIG_Diag_Inputs_Channel_2.Diag_Input[0] <-> DIG Diag Inputs  Channel 2/Diag Input 1
//     PlcTask Inputs/GVL_iXlinker.EtherCAT_Master_EPPxxxx.Beckhoff_EPP2xxx.Beckhoff_EPP2xxxEK1122.A_0076_EPP2816_0008_0017.DIG_Diag_Inputs_Channel_2.Diag_Input[1] <-> DIG Diag Inputs  Channel 2/Diag Input 2
//     PlcTask Inputs/GVL_iXlinker.EtherCAT_Master_EPPxxxx.Beckhoff_EPP2xxx.Beckhoff_EPP2xxxEK1122.A_0076_EPP2816_0008_0017.DIG_Diag_Inputs_Channel_2.Diag_Input[2] <-> DIG Diag Inputs  Channel 2/Diag Input 3
//     PlcTask Inputs/GVL_iXlinker.EtherCAT_Master_EPPxxxx.Beckhoff_EPP2xxx.Beckhoff_EPP2xxxEK1122.A_0076_EPP2816_0008_0017.DIG_Diag_Inputs_Channel_2.Diag_Input[3] <-> DIG Diag Inputs  Channel 2/Diag Input 4
//     PlcTask Inputs/GVL_iXlinker.EtherCAT_Master_EPPxxxx.Beckhoff_EPP2xxx.Beckhoff_EPP2xxxEK1122.A_0076_EPP2816_0008_0017.DIG_Diag_Inputs_Channel_2.Diag_Input[4] <-> DIG Diag Inputs  Channel 2/Diag Input 5
//     PlcTask Inputs/GVL_iXlinker.EtherCAT_Master_EPPxxxx.Beckhoff_EPP2xxx.Beckhoff_EPP2xxxEK1122.A_0076_EPP2816_0008_0017.DIG_Diag_Inputs_Channel_2.Diag_Input[5] <-> DIG Diag Inputs  Channel 2/Diag Input 6
//     PlcTask Inputs/GVL_iXlinker.EtherCAT_Master_EPPxxxx.Beckhoff_EPP2xxx.Beckhoff_EPP2xxxEK1122.A_0076_EPP2816_0008_0017.DIG_Diag_Inputs_Channel_2.Diag_Input[6] <-> DIG Diag Inputs  Channel 2/Diag Input 7
//     PlcTask Inputs/GVL_iXlinker.EtherCAT_Master_EPPxxxx.Beckhoff_EPP2xxx.Beckhoff_EPP2xxxEK1122.A_0076_EPP2816_0008_0017.DIG_Diag_Inputs_Channel_2.Diag_Input[7] <-> DIG Diag Inputs  Channel 2/Diag Input 8
//     PlcTask Inputs/GVL_iXlinker.EtherCAT_Master_EPPxxxx.Beckhoff_EPP2xxx.Beckhoff_EPP2xxxEK1122.A_0076_EPP2816_0008_0017.DIG_Inputs_Device.Safe_state_active <-> DIG Inputs Device/Safe state active
//     PlcTask Inputs/GVL_iXlinker.EtherCAT_Master_EPPxxxx.Beckhoff_EPP2xxx.Beckhoff_EPP2xxxEK1122.A_0076_EPP2816_0008_0017.DIG_Inputs_Device.Error_channel[0] <-> DIG Inputs Device/Error channel 1
//     PlcTask Inputs/GVL_iXlinker.EtherCAT_Master_EPPxxxx.Beckhoff_EPP2xxx.Beckhoff_EPP2xxxEK1122.A_0076_EPP2816_0008_0017.DIG_Inputs_Device.Error_channel[1] <-> DIG Inputs Device/Error channel 2
//     PlcTask Inputs/GVL_iXlinker.EtherCAT_Master_EPPxxxx.Beckhoff_EPP2xxx.Beckhoff_EPP2xxxEK1122.A_0076_EPP2816_0008_0017.DIG_Inputs_Device.Sync_error <-> DIG Inputs Device/Sync error
//     PlcTask Inputs/GVL_iXlinker.EtherCAT_Master_EPPxxxx.Beckhoff_EPP2xxx.Beckhoff_EPP2xxxEK1122.A_0076_EPP2816_0008_0017.DIG_Inputs_Device.TxPDO_Toggle <-> DIG Inputs Device/TxPDO Toggle
//     PlcTask Outputs/GVL_iXlinker.EtherCAT_Master_EPPxxxx.Beckhoff_EPP2xxx.Beckhoff_EPP2xxxEK1122.A_0076_EPP2816_0008_0017.DIG_Outputs_Channel_1.Output[0] <-> DIG Outputs Channel 1/Output 1
//     PlcTask Outputs/GVL_iXlinker.EtherCAT_Master_EPPxxxx.Beckhoff_EPP2xxx.Beckhoff_EPP2xxxEK1122.A_0076_EPP2816_0008_0017.DIG_Outputs_Channel_1.Output[1] <-> DIG Outputs Channel 1/Output 2
//     PlcTask Outputs/GVL_iXlinker.EtherCAT_Master_EPPxxxx.Beckhoff_EPP2xxx.Beckhoff_EPP2xxxEK1122.A_0076_EPP2816_0008_0017.DIG_Outputs_Channel_1.Output[2] <-> DIG Outputs Channel 1/Output 3
//     PlcTask Outputs/GVL_iXlinker.EtherCAT_Master_EPPxxxx.Beckhoff_EPP2xxx.Beckhoff_EPP2xxxEK1122.A_0076_EPP2816_0008_0017.DIG_Outputs_Channel_1.Output[3] <-> DIG Outputs Channel 1/Output 4
//     PlcTask Outputs/GVL_iXlinker.EtherCAT_Master_EPPxxxx.Beckhoff_EPP2xxx.Beckhoff_EPP2xxxEK1122.A_0076_EPP2816_0008_0017.DIG_Outputs_Channel_1.Output[4] <-> DIG Outputs Channel 1/Output 5
//     PlcTask Outputs/GVL_iXlinker.EtherCAT_Master_EPPxxxx.Beckhoff_EPP2xxx.Beckhoff_EPP2xxxEK1122.A_0076_EPP2816_0008_0017.DIG_Outputs_Channel_1.Output[5] <-> DIG Outputs Channel 1/Output 6
//     PlcTask Outputs/GVL_iXlinker.EtherCAT_Master_EPPxxxx.Beckhoff_EPP2xxx.Beckhoff_EPP2xxxEK1122.A_0076_EPP2816_0008_0017.DIG_Outputs_Channel_1.Output[6] <-> DIG Outputs Channel 1/Output 7
//     PlcTask Outputs/GVL_iXlinker.EtherCAT_Master_EPPxxxx.Beckhoff_EPP2xxx.Beckhoff_EPP2xxxEK1122.A_0076_EPP2816_0008_0017.DIG_Outputs_Channel_1.Output[7] <-> DIG Outputs Channel 1/Output 8
//     PlcTask Outputs/GVL_iXlinker.EtherCAT_Master_EPPxxxx.Beckhoff_EPP2xxx.Beckhoff_EPP2xxxEK1122.A_0076_EPP2816_0008_0017.DIG_Outputs_Channel_2.Output[0] <-> DIG Outputs Channel 2/Output 1
//     PlcTask Outputs/GVL_iXlinker.EtherCAT_Master_EPPxxxx.Beckhoff_EPP2xxx.Beckhoff_EPP2xxxEK1122.A_0076_EPP2816_0008_0017.DIG_Outputs_Channel_2.Output[1] <-> DIG Outputs Channel 2/Output 2
//     PlcTask Outputs/GVL_iXlinker.EtherCAT_Master_EPPxxxx.Beckhoff_EPP2xxx.Beckhoff_EPP2xxxEK1122.A_0076_EPP2816_0008_0017.DIG_Outputs_Channel_2.Output[2] <-> DIG Outputs Channel 2/Output 3
//     PlcTask Outputs/GVL_iXlinker.EtherCAT_Master_EPPxxxx.Beckhoff_EPP2xxx.Beckhoff_EPP2xxxEK1122.A_0076_EPP2816_0008_0017.DIG_Outputs_Channel_2.Output[3] <-> DIG Outputs Channel 2/Output 4
//     PlcTask Outputs/GVL_iXlinker.EtherCAT_Master_EPPxxxx.Beckhoff_EPP2xxx.Beckhoff_EPP2xxxEK1122.A_0076_EPP2816_0008_0017.DIG_Outputs_Channel_2.Output[4] <-> DIG Outputs Channel 2/Output 5
//     PlcTask Outputs/GVL_iXlinker.EtherCAT_Master_EPPxxxx.Beckhoff_EPP2xxx.Beckhoff_EPP2xxxEK1122.A_0076_EPP2816_0008_0017.DIG_Outputs_Channel_2.Output[5] <-> DIG Outputs Channel 2/Output 6
//     PlcTask Outputs/GVL_iXlinker.EtherCAT_Master_EPPxxxx.Beckhoff_EPP2xxx.Beckhoff_EPP2xxxEK1122.A_0076_EPP2816_0008_0017.DIG_Outputs_Channel_2.Output[6] <-> DIG Outputs Channel 2/Output 7
//     PlcTask Outputs/GVL_iXlinker.EtherCAT_Master_EPPxxxx.Beckhoff_EPP2xxx.Beckhoff_EPP2xxxEK1122.A_0076_EPP2816_0008_0017.DIG_Outputs_Channel_2.Output[7] <-> DIG Outputs Channel 2/Output 8
//     PlcTask Outputs/GVL_iXlinker.EtherCAT_Master_EPPxxxx.Beckhoff_EPP2xxx.Beckhoff_EPP2xxxEK1122.A_0076_EPP2816_0008_0017.DIG_Outputs_Device.Set_safe_state <-> DIG Outputs Device/Set safe state
//     PlcTask Outputs/GVL_iXlinker.EtherCAT_Master_EPPxxxx.Beckhoff_EPP2xxx.Beckhoff_EPP2xxxEK1122.A_0076_EPP2816_0008_0017.DIG_Outputs_Device.Reset_outputs <-> DIG Outputs Device/Reset outputs
//     PlcTask Inputs/GVL_iXlinker.EtherCAT_Master_EPPxxxx.Beckhoff_EPP2xxx.Beckhoff_EPP2xxxEK1122.A_0076_EPP2816_0008_0017.WcState.WcState <-> WcState/WcState
//     PlcTask Inputs/GVL_iXlinker.EtherCAT_Master_EPPxxxx.Beckhoff_EPP2xxx.Beckhoff_EPP2xxxEK1122.A_0076_EPP2816_0008_0017.WcState.InputToggle <-> WcState/InputToggle
//     PlcTask Inputs/GVL_iXlinker.EtherCAT_Master_EPPxxxx.Beckhoff_EPP2xxx.Beckhoff_EPP2xxxEK1122.A_0076_EPP2816_0008_0017.InfoData.AdsAddr <-> InfoData/AdsAddr
//     PlcTask Inputs/GVL_iXlinker.EtherCAT_Master_EPPxxxx.Beckhoff_EPP2xxx.Beckhoff_EPP2xxxEK1122.A_0076_EPP2816_0008_0017.InfoData.State <-> InfoData/State
//   PLC/PLC Instance <-> EtherCAT Master EPPxxxx/Beckhoff EPP2xxx/Beckhoff EPP2xxxEK1122/A_0077(EPP2816-0008-0018)
//     PlcTask Inputs/GVL_iXlinker.EtherCAT_Master_EPPxxxx.Beckhoff_EPP2xxx.Beckhoff_EPP2xxxEK1122.A_0077_EPP2816_0008_0018.DIG_Diag_Inputs_Channel_1.Diag_Input[0] <-> DIG Diag Inputs  Channel 1/Diag Input 1
//     PlcTask Inputs/GVL_iXlinker.EtherCAT_Master_EPPxxxx.Beckhoff_EPP2xxx.Beckhoff_EPP2xxxEK1122.A_0077_EPP2816_0008_0018.DIG_Diag_Inputs_Channel_1.Diag_Input[1] <-> DIG Diag Inputs  Channel 1/Diag Input 2
//     PlcTask Inputs/GVL_iXlinker.EtherCAT_Master_EPPxxxx.Beckhoff_EPP2xxx.Beckhoff_EPP2xxxEK1122.A_0077_EPP2816_0008_0018.DIG_Diag_Inputs_Channel_1.Diag_Input[2] <-> DIG Diag Inputs  Channel 1/Diag Input 3
//     PlcTask Inputs/GVL_iXlinker.EtherCAT_Master_EPPxxxx.Beckhoff_EPP2xxx.Beckhoff_EPP2xxxEK1122.A_0077_EPP2816_0008_0018.DIG_Diag_Inputs_Channel_1.Diag_Input[3] <-> DIG Diag Inputs  Channel 1/Diag Input 4
//     PlcTask Inputs/GVL_iXlinker.EtherCAT_Master_EPPxxxx.Beckhoff_EPP2xxx.Beckhoff_EPP2xxxEK1122.A_0077_EPP2816_0008_0018.DIG_Diag_Inputs_Channel_1.Diag_Input[4] <-> DIG Diag Inputs  Channel 1/Diag Input 5
//     PlcTask Inputs/GVL_iXlinker.EtherCAT_Master_EPPxxxx.Beckhoff_EPP2xxx.Beckhoff_EPP2xxxEK1122.A_0077_EPP2816_0008_0018.DIG_Diag_Inputs_Channel_1.Diag_Input[5] <-> DIG Diag Inputs  Channel 1/Diag Input 6
//     PlcTask Inputs/GVL_iXlinker.EtherCAT_Master_EPPxxxx.Beckhoff_EPP2xxx.Beckhoff_EPP2xxxEK1122.A_0077_EPP2816_0008_0018.DIG_Diag_Inputs_Channel_1.Diag_Input[6] <-> DIG Diag Inputs  Channel 1/Diag Input 7
//     PlcTask Inputs/GVL_iXlinker.EtherCAT_Master_EPPxxxx.Beckhoff_EPP2xxx.Beckhoff_EPP2xxxEK1122.A_0077_EPP2816_0008_0018.DIG_Diag_Inputs_Channel_1.Diag_Input[7] <-> DIG Diag Inputs  Channel 1/Diag Input 8
//     PlcTask Inputs/GVL_iXlinker.EtherCAT_Master_EPPxxxx.Beckhoff_EPP2xxx.Beckhoff_EPP2xxxEK1122.A_0077_EPP2816_0008_0018.DIG_Diag_Inputs_Channel_2.Diag_Input[0] <-> DIG Diag Inputs  Channel 2/Diag Input 1
//     PlcTask Inputs/GVL_iXlinker.EtherCAT_Master_EPPxxxx.Beckhoff_EPP2xxx.Beckhoff_EPP2xxxEK1122.A_0077_EPP2816_0008_0018.DIG_Diag_Inputs_Channel_2.Diag_Input[1] <-> DIG Diag Inputs  Channel 2/Diag Input 2
//     PlcTask Inputs/GVL_iXlinker.EtherCAT_Master_EPPxxxx.Beckhoff_EPP2xxx.Beckhoff_EPP2xxxEK1122.A_0077_EPP2816_0008_0018.DIG_Diag_Inputs_Channel_2.Diag_Input[2] <-> DIG Diag Inputs  Channel 2/Diag Input 3
//     PlcTask Inputs/GVL_iXlinker.EtherCAT_Master_EPPxxxx.Beckhoff_EPP2xxx.Beckhoff_EPP2xxxEK1122.A_0077_EPP2816_0008_0018.DIG_Diag_Inputs_Channel_2.Diag_Input[3] <-> DIG Diag Inputs  Channel 2/Diag Input 4
//     PlcTask Inputs/GVL_iXlinker.EtherCAT_Master_EPPxxxx.Beckhoff_EPP2xxx.Beckhoff_EPP2xxxEK1122.A_0077_EPP2816_0008_0018.DIG_Diag_Inputs_Channel_2.Diag_Input[4] <-> DIG Diag Inputs  Channel 2/Diag Input 5
//     PlcTask Inputs/GVL_iXlinker.EtherCAT_Master_EPPxxxx.Beckhoff_EPP2xxx.Beckhoff_EPP2xxxEK1122.A_0077_EPP2816_0008_0018.DIG_Diag_Inputs_Channel_2.Diag_Input[5] <-> DIG Diag Inputs  Channel 2/Diag Input 6
//     PlcTask Inputs/GVL_iXlinker.EtherCAT_Master_EPPxxxx.Beckhoff_EPP2xxx.Beckhoff_EPP2xxxEK1122.A_0077_EPP2816_0008_0018.DIG_Diag_Inputs_Channel_2.Diag_Input[6] <-> DIG Diag Inputs  Channel 2/Diag Input 7
//     PlcTask Inputs/GVL_iXlinker.EtherCAT_Master_EPPxxxx.Beckhoff_EPP2xxx.Beckhoff_EPP2xxxEK1122.A_0077_EPP2816_0008_0018.DIG_Diag_Inputs_Channel_2.Diag_Input[7] <-> DIG Diag Inputs  Channel 2/Diag Input 8
//     PlcTask Inputs/GVL_iXlinker.EtherCAT_Master_EPPxxxx.Beckhoff_EPP2xxx.Beckhoff_EPP2xxxEK1122.A_0077_EPP2816_0008_0018.DIG_Inputs_Device.Safe_state_active <-> DIG Inputs Device/Safe state active
//     PlcTask Inputs/GVL_iXlinker.EtherCAT_Master_EPPxxxx.Beckhoff_EPP2xxx.Beckhoff_EPP2xxxEK1122.A_0077_EPP2816_0008_0018.DIG_Inputs_Device.Error_channel[0] <-> DIG Inputs Device/Error channel 1
//     PlcTask Inputs/GVL_iXlinker.EtherCAT_Master_EPPxxxx.Beckhoff_EPP2xxx.Beckhoff_EPP2xxxEK1122.A_0077_EPP2816_0008_0018.DIG_Inputs_Device.Error_channel[1] <-> DIG Inputs Device/Error channel 2
//     PlcTask Inputs/GVL_iXlinker.EtherCAT_Master_EPPxxxx.Beckhoff_EPP2xxx.Beckhoff_EPP2xxxEK1122.A_0077_EPP2816_0008_0018.DIG_Inputs_Device.Sync_error <-> DIG Inputs Device/Sync error
//     PlcTask Inputs/GVL_iXlinker.EtherCAT_Master_EPPxxxx.Beckhoff_EPP2xxx.Beckhoff_EPP2xxxEK1122.A_0077_EPP2816_0008_0018.DIG_Inputs_Device.TxPDO_Toggle <-> DIG Inputs Device/TxPDO Toggle
//     PlcTask Outputs/GVL_iXlinker.EtherCAT_Master_EPPxxxx.Beckhoff_EPP2xxx.Beckhoff_EPP2xxxEK1122.A_0077_EPP2816_0008_0018.DIG_Outputs_Channel_1.Output[0] <-> DIG Outputs Channel 1/Output 1
//     PlcTask Outputs/GVL_iXlinker.EtherCAT_Master_EPPxxxx.Beckhoff_EPP2xxx.Beckhoff_EPP2xxxEK1122.A_0077_EPP2816_0008_0018.DIG_Outputs_Channel_1.Output[1] <-> DIG Outputs Channel 1/Output 2
//     PlcTask Outputs/GVL_iXlinker.EtherCAT_Master_EPPxxxx.Beckhoff_EPP2xxx.Beckhoff_EPP2xxxEK1122.A_0077_EPP2816_0008_0018.DIG_Outputs_Channel_1.Output[2] <-> DIG Outputs Channel 1/Output 3
//     PlcTask Outputs/GVL_iXlinker.EtherCAT_Master_EPPxxxx.Beckhoff_EPP2xxx.Beckhoff_EPP2xxxEK1122.A_0077_EPP2816_0008_0018.DIG_Outputs_Channel_1.Output[3] <-> DIG Outputs Channel 1/Output 4
//     PlcTask Outputs/GVL_iXlinker.EtherCAT_Master_EPPxxxx.Beckhoff_EPP2xxx.Beckhoff_EPP2xxxEK1122.A_0077_EPP2816_0008_0018.DIG_Outputs_Channel_1.Output[4] <-> DIG Outputs Channel 1/Output 5
//     PlcTask Outputs/GVL_iXlinker.EtherCAT_Master_EPPxxxx.Beckhoff_EPP2xxx.Beckhoff_EPP2xxxEK1122.A_0077_EPP2816_0008_0018.DIG_Outputs_Channel_1.Output[5] <-> DIG Outputs Channel 1/Output 6
//     PlcTask Outputs/GVL_iXlinker.EtherCAT_Master_EPPxxxx.Beckhoff_EPP2xxx.Beckhoff_EPP2xxxEK1122.A_0077_EPP2816_0008_0018.DIG_Outputs_Channel_1.Output[6] <-> DIG Outputs Channel 1/Output 7
//     PlcTask Outputs/GVL_iXlinker.EtherCAT_Master_EPPxxxx.Beckhoff_EPP2xxx.Beckhoff_EPP2xxxEK1122.A_0077_EPP2816_0008_0018.DIG_Outputs_Channel_1.Output[7] <-> DIG Outputs Channel 1/Output 8
//     PlcTask Outputs/GVL_iXlinker.EtherCAT_Master_EPPxxxx.Beckhoff_EPP2xxx.Beckhoff_EPP2xxxEK1122.A_0077_EPP2816_0008_0018.DIG_Outputs_Channel_2.Output[0] <-> DIG Outputs Channel 2/Output 1
//     PlcTask Outputs/GVL_iXlinker.EtherCAT_Master_EPPxxxx.Beckhoff_EPP2xxx.Beckhoff_EPP2xxxEK1122.A_0077_EPP2816_0008_0018.DIG_Outputs_Channel_2.Output[1] <-> DIG Outputs Channel 2/Output 2
//     PlcTask Outputs/GVL_iXlinker.EtherCAT_Master_EPPxxxx.Beckhoff_EPP2xxx.Beckhoff_EPP2xxxEK1122.A_0077_EPP2816_0008_0018.DIG_Outputs_Channel_2.Output[2] <-> DIG Outputs Channel 2/Output 3
//     PlcTask Outputs/GVL_iXlinker.EtherCAT_Master_EPPxxxx.Beckhoff_EPP2xxx.Beckhoff_EPP2xxxEK1122.A_0077_EPP2816_0008_0018.DIG_Outputs_Channel_2.Output[3] <-> DIG Outputs Channel 2/Output 4
//     PlcTask Outputs/GVL_iXlinker.EtherCAT_Master_EPPxxxx.Beckhoff_EPP2xxx.Beckhoff_EPP2xxxEK1122.A_0077_EPP2816_0008_0018.DIG_Outputs_Channel_2.Output[4] <-> DIG Outputs Channel 2/Output 5
//     PlcTask Outputs/GVL_iXlinker.EtherCAT_Master_EPPxxxx.Beckhoff_EPP2xxx.Beckhoff_EPP2xxxEK1122.A_0077_EPP2816_0008_0018.DIG_Outputs_Channel_2.Output[5] <-> DIG Outputs Channel 2/Output 6
//     PlcTask Outputs/GVL_iXlinker.EtherCAT_Master_EPPxxxx.Beckhoff_EPP2xxx.Beckhoff_EPP2xxxEK1122.A_0077_EPP2816_0008_0018.DIG_Outputs_Channel_2.Output[6] <-> DIG Outputs Channel 2/Output 7
//     PlcTask Outputs/GVL_iXlinker.EtherCAT_Master_EPPxxxx.Beckhoff_EPP2xxx.Beckhoff_EPP2xxxEK1122.A_0077_EPP2816_0008_0018.DIG_Outputs_Channel_2.Output[7] <-> DIG Outputs Channel 2/Output 8
//     PlcTask Outputs/GVL_iXlinker.EtherCAT_Master_EPPxxxx.Beckhoff_EPP2xxx.Beckhoff_EPP2xxxEK1122.A_0077_EPP2816_0008_0018.DIG_Outputs_Device.Set_safe_state <-> DIG Outputs Device/Set safe state
//     PlcTask Outputs/GVL_iXlinker.EtherCAT_Master_EPPxxxx.Beckhoff_EPP2xxx.Beckhoff_EPP2xxxEK1122.A_0077_EPP2816_0008_0018.DIG_Outputs_Device.Reset_outputs <-> DIG Outputs Device/Reset outputs
//     PlcTask Inputs/GVL_iXlinker.EtherCAT_Master_EPPxxxx.Beckhoff_EPP2xxx.Beckhoff_EPP2xxxEK1122.A_0077_EPP2816_0008_0018.WcState.WcState <-> WcState/WcState
//     PlcTask Inputs/GVL_iXlinker.EtherCAT_Master_EPPxxxx.Beckhoff_EPP2xxx.Beckhoff_EPP2xxxEK1122.A_0077_EPP2816_0008_0018.WcState.InputToggle <-> WcState/InputToggle
//     PlcTask Inputs/GVL_iXlinker.EtherCAT_Master_EPPxxxx.Beckhoff_EPP2xxx.Beckhoff_EPP2xxxEK1122.A_0077_EPP2816_0008_0018.InfoData.AdsAddr <-> InfoData/AdsAddr
//     PlcTask Inputs/GVL_iXlinker.EtherCAT_Master_EPPxxxx.Beckhoff_EPP2xxx.Beckhoff_EPP2xxxEK1122.A_0077_EPP2816_0008_0018.InfoData.State <-> InfoData/State
//   PLC/PLC Instance <-> EtherCAT Master EPPxxxx/Beckhoff EPP2xxx/Beckhoff EPP2xxxEK1122/A_0078(EPP2816-0010-0016)
//     PlcTask Inputs/GVL_iXlinker.EtherCAT_Master_EPPxxxx.Beckhoff_EPP2xxx.Beckhoff_EPP2xxxEK1122.A_0078_EPP2816_0010_0016.DIG_Diag_Inputs_Channel_1.Diag_Input[0] <-> DIG Diag Inputs  Channel 1/Diag Input 1
//     PlcTask Inputs/GVL_iXlinker.EtherCAT_Master_EPPxxxx.Beckhoff_EPP2xxx.Beckhoff_EPP2xxxEK1122.A_0078_EPP2816_0010_0016.DIG_Diag_Inputs_Channel_1.Diag_Input[1] <-> DIG Diag Inputs  Channel 1/Diag Input 2
//     PlcTask Inputs/GVL_iXlinker.EtherCAT_Master_EPPxxxx.Beckhoff_EPP2xxx.Beckhoff_EPP2xxxEK1122.A_0078_EPP2816_0010_0016.DIG_Diag_Inputs_Channel_1.Diag_Input[2] <-> DIG Diag Inputs  Channel 1/Diag Input 3
//     PlcTask Inputs/GVL_iXlinker.EtherCAT_Master_EPPxxxx.Beckhoff_EPP2xxx.Beckhoff_EPP2xxxEK1122.A_0078_EPP2816_0010_0016.DIG_Diag_Inputs_Channel_1.Diag_Input[3] <-> DIG Diag Inputs  Channel 1/Diag Input 4
//     PlcTask Inputs/GVL_iXlinker.EtherCAT_Master_EPPxxxx.Beckhoff_EPP2xxx.Beckhoff_EPP2xxxEK1122.A_0078_EPP2816_0010_0016.DIG_Diag_Inputs_Channel_1.Diag_Input[4] <-> DIG Diag Inputs  Channel 1/Diag Input 5
//     PlcTask Inputs/GVL_iXlinker.EtherCAT_Master_EPPxxxx.Beckhoff_EPP2xxx.Beckhoff_EPP2xxxEK1122.A_0078_EPP2816_0010_0016.DIG_Diag_Inputs_Channel_1.Diag_Input[5] <-> DIG Diag Inputs  Channel 1/Diag Input 6
//     PlcTask Inputs/GVL_iXlinker.EtherCAT_Master_EPPxxxx.Beckhoff_EPP2xxx.Beckhoff_EPP2xxxEK1122.A_0078_EPP2816_0010_0016.DIG_Diag_Inputs_Channel_1.Diag_Input[6] <-> DIG Diag Inputs  Channel 1/Diag Input 7
//     PlcTask Inputs/GVL_iXlinker.EtherCAT_Master_EPPxxxx.Beckhoff_EPP2xxx.Beckhoff_EPP2xxxEK1122.A_0078_EPP2816_0010_0016.DIG_Diag_Inputs_Channel_1.Diag_Input[7] <-> DIG Diag Inputs  Channel 1/Diag Input 8
//     PlcTask Inputs/GVL_iXlinker.EtherCAT_Master_EPPxxxx.Beckhoff_EPP2xxx.Beckhoff_EPP2xxxEK1122.A_0078_EPP2816_0010_0016.DIG_Diag_Inputs_Channel_2.Diag_Input[0] <-> DIG Diag Inputs  Channel 2/Diag Input 1
//     PlcTask Inputs/GVL_iXlinker.EtherCAT_Master_EPPxxxx.Beckhoff_EPP2xxx.Beckhoff_EPP2xxxEK1122.A_0078_EPP2816_0010_0016.DIG_Diag_Inputs_Channel_2.Diag_Input[1] <-> DIG Diag Inputs  Channel 2/Diag Input 2
//     PlcTask Inputs/GVL_iXlinker.EtherCAT_Master_EPPxxxx.Beckhoff_EPP2xxx.Beckhoff_EPP2xxxEK1122.A_0078_EPP2816_0010_0016.DIG_Diag_Inputs_Channel_2.Diag_Input[2] <-> DIG Diag Inputs  Channel 2/Diag Input 3
//     PlcTask Inputs/GVL_iXlinker.EtherCAT_Master_EPPxxxx.Beckhoff_EPP2xxx.Beckhoff_EPP2xxxEK1122.A_0078_EPP2816_0010_0016.DIG_Diag_Inputs_Channel_2.Diag_Input[3] <-> DIG Diag Inputs  Channel 2/Diag Input 4
//     PlcTask Inputs/GVL_iXlinker.EtherCAT_Master_EPPxxxx.Beckhoff_EPP2xxx.Beckhoff_EPP2xxxEK1122.A_0078_EPP2816_0010_0016.DIG_Diag_Inputs_Channel_2.Diag_Input[4] <-> DIG Diag Inputs  Channel 2/Diag Input 5
//     PlcTask Inputs/GVL_iXlinker.EtherCAT_Master_EPPxxxx.Beckhoff_EPP2xxx.Beckhoff_EPP2xxxEK1122.A_0078_EPP2816_0010_0016.DIG_Diag_Inputs_Channel_2.Diag_Input[5] <-> DIG Diag Inputs  Channel 2/Diag Input 6
//     PlcTask Inputs/GVL_iXlinker.EtherCAT_Master_EPPxxxx.Beckhoff_EPP2xxx.Beckhoff_EPP2xxxEK1122.A_0078_EPP2816_0010_0016.DIG_Diag_Inputs_Channel_2.Diag_Input[6] <-> DIG Diag Inputs  Channel 2/Diag Input 7
//     PlcTask Inputs/GVL_iXlinker.EtherCAT_Master_EPPxxxx.Beckhoff_EPP2xxx.Beckhoff_EPP2xxxEK1122.A_0078_EPP2816_0010_0016.DIG_Diag_Inputs_Channel_2.Diag_Input[7] <-> DIG Diag Inputs  Channel 2/Diag Input 8
//     PlcTask Inputs/GVL_iXlinker.EtherCAT_Master_EPPxxxx.Beckhoff_EPP2xxx.Beckhoff_EPP2xxxEK1122.A_0078_EPP2816_0010_0016.DIG_Inputs_Device.Safe_state_active <-> DIG Inputs Device/Safe state active
//     PlcTask Inputs/GVL_iXlinker.EtherCAT_Master_EPPxxxx.Beckhoff_EPP2xxx.Beckhoff_EPP2xxxEK1122.A_0078_EPP2816_0010_0016.DIG_Inputs_Device.Error_channel[0] <-> DIG Inputs Device/Error channel 1
//     PlcTask Inputs/GVL_iXlinker.EtherCAT_Master_EPPxxxx.Beckhoff_EPP2xxx.Beckhoff_EPP2xxxEK1122.A_0078_EPP2816_0010_0016.DIG_Inputs_Device.Error_channel[1] <-> DIG Inputs Device/Error channel 2
//     PlcTask Inputs/GVL_iXlinker.EtherCAT_Master_EPPxxxx.Beckhoff_EPP2xxx.Beckhoff_EPP2xxxEK1122.A_0078_EPP2816_0010_0016.DIG_Inputs_Device.Sync_error <-> DIG Inputs Device/Sync error
//     PlcTask Inputs/GVL_iXlinker.EtherCAT_Master_EPPxxxx.Beckhoff_EPP2xxx.Beckhoff_EPP2xxxEK1122.A_0078_EPP2816_0010_0016.DIG_Inputs_Device.TxPDO_Toggle <-> DIG Inputs Device/TxPDO Toggle
//     PlcTask Outputs/GVL_iXlinker.EtherCAT_Master_EPPxxxx.Beckhoff_EPP2xxx.Beckhoff_EPP2xxxEK1122.A_0078_EPP2816_0010_0016.DIG_Outputs_Channel_1.Output[0] <-> DIG Outputs Channel 1/Output 1
//     PlcTask Outputs/GVL_iXlinker.EtherCAT_Master_EPPxxxx.Beckhoff_EPP2xxx.Beckhoff_EPP2xxxEK1122.A_0078_EPP2816_0010_0016.DIG_Outputs_Channel_1.Output[1] <-> DIG Outputs Channel 1/Output 2
//     PlcTask Outputs/GVL_iXlinker.EtherCAT_Master_EPPxxxx.Beckhoff_EPP2xxx.Beckhoff_EPP2xxxEK1122.A_0078_EPP2816_0010_0016.DIG_Outputs_Channel_1.Output[2] <-> DIG Outputs Channel 1/Output 3
//     PlcTask Outputs/GVL_iXlinker.EtherCAT_Master_EPPxxxx.Beckhoff_EPP2xxx.Beckhoff_EPP2xxxEK1122.A_0078_EPP2816_0010_0016.DIG_Outputs_Channel_1.Output[3] <-> DIG Outputs Channel 1/Output 4
//     PlcTask Outputs/GVL_iXlinker.EtherCAT_Master_EPPxxxx.Beckhoff_EPP2xxx.Beckhoff_EPP2xxxEK1122.A_0078_EPP2816_0010_0016.DIG_Outputs_Channel_1.Output[4] <-> DIG Outputs Channel 1/Output 5
//     PlcTask Outputs/GVL_iXlinker.EtherCAT_Master_EPPxxxx.Beckhoff_EPP2xxx.Beckhoff_EPP2xxxEK1122.A_0078_EPP2816_0010_0016.DIG_Outputs_Channel_1.Output[5] <-> DIG Outputs Channel 1/Output 6
//     PlcTask Outputs/GVL_iXlinker.EtherCAT_Master_EPPxxxx.Beckhoff_EPP2xxx.Beckhoff_EPP2xxxEK1122.A_0078_EPP2816_0010_0016.DIG_Outputs_Channel_1.Output[6] <-> DIG Outputs Channel 1/Output 7
//     PlcTask Outputs/GVL_iXlinker.EtherCAT_Master_EPPxxxx.Beckhoff_EPP2xxx.Beckhoff_EPP2xxxEK1122.A_0078_EPP2816_0010_0016.DIG_Outputs_Channel_1.Output[7] <-> DIG Outputs Channel 1/Output 8
//     PlcTask Outputs/GVL_iXlinker.EtherCAT_Master_EPPxxxx.Beckhoff_EPP2xxx.Beckhoff_EPP2xxxEK1122.A_0078_EPP2816_0010_0016.DIG_Outputs_Channel_2.Output[0] <-> DIG Outputs Channel 2/Output 1
//     PlcTask Outputs/GVL_iXlinker.EtherCAT_Master_EPPxxxx.Beckhoff_EPP2xxx.Beckhoff_EPP2xxxEK1122.A_0078_EPP2816_0010_0016.DIG_Outputs_Channel_2.Output[1] <-> DIG Outputs Channel 2/Output 2
//     PlcTask Outputs/GVL_iXlinker.EtherCAT_Master_EPPxxxx.Beckhoff_EPP2xxx.Beckhoff_EPP2xxxEK1122.A_0078_EPP2816_0010_0016.DIG_Outputs_Channel_2.Output[2] <-> DIG Outputs Channel 2/Output 3
//     PlcTask Outputs/GVL_iXlinker.EtherCAT_Master_EPPxxxx.Beckhoff_EPP2xxx.Beckhoff_EPP2xxxEK1122.A_0078_EPP2816_0010_0016.DIG_Outputs_Channel_2.Output[3] <-> DIG Outputs Channel 2/Output 4
//     PlcTask Outputs/GVL_iXlinker.EtherCAT_Master_EPPxxxx.Beckhoff_EPP2xxx.Beckhoff_EPP2xxxEK1122.A_0078_EPP2816_0010_0016.DIG_Outputs_Channel_2.Output[4] <-> DIG Outputs Channel 2/Output 5
//     PlcTask Outputs/GVL_iXlinker.EtherCAT_Master_EPPxxxx.Beckhoff_EPP2xxx.Beckhoff_EPP2xxxEK1122.A_0078_EPP2816_0010_0016.DIG_Outputs_Channel_2.Output[5] <-> DIG Outputs Channel 2/Output 6
//     PlcTask Outputs/GVL_iXlinker.EtherCAT_Master_EPPxxxx.Beckhoff_EPP2xxx.Beckhoff_EPP2xxxEK1122.A_0078_EPP2816_0010_0016.DIG_Outputs_Channel_2.Output[6] <-> DIG Outputs Channel 2/Output 7
//     PlcTask Outputs/GVL_iXlinker.EtherCAT_Master_EPPxxxx.Beckhoff_EPP2xxx.Beckhoff_EPP2xxxEK1122.A_0078_EPP2816_0010_0016.DIG_Outputs_Channel_2.Output[7] <-> DIG Outputs Channel 2/Output 8
//     PlcTask Outputs/GVL_iXlinker.EtherCAT_Master_EPPxxxx.Beckhoff_EPP2xxx.Beckhoff_EPP2xxxEK1122.A_0078_EPP2816_0010_0016.DIG_Outputs_Device.Set_safe_state <-> DIG Outputs Device/Set safe state
//     PlcTask Outputs/GVL_iXlinker.EtherCAT_Master_EPPxxxx.Beckhoff_EPP2xxx.Beckhoff_EPP2xxxEK1122.A_0078_EPP2816_0010_0016.DIG_Outputs_Device.Reset_outputs <-> DIG Outputs Device/Reset outputs
//     PlcTask Inputs/GVL_iXlinker.EtherCAT_Master_EPPxxxx.Beckhoff_EPP2xxx.Beckhoff_EPP2xxxEK1122.A_0078_EPP2816_0010_0016.WcState.WcState <-> WcState/WcState
//     PlcTask Inputs/GVL_iXlinker.EtherCAT_Master_EPPxxxx.Beckhoff_EPP2xxx.Beckhoff_EPP2xxxEK1122.A_0078_EPP2816_0010_0016.WcState.InputToggle <-> WcState/InputToggle
//     PlcTask Inputs/GVL_iXlinker.EtherCAT_Master_EPPxxxx.Beckhoff_EPP2xxx.Beckhoff_EPP2xxxEK1122.A_0078_EPP2816_0010_0016.InfoData.AdsAddr <-> InfoData/AdsAddr
//     PlcTask Inputs/GVL_iXlinker.EtherCAT_Master_EPPxxxx.Beckhoff_EPP2xxx.Beckhoff_EPP2xxxEK1122.A_0078_EPP2816_0010_0016.InfoData.State <-> InfoData/State
//   PLC/PLC Instance <-> EtherCAT Master EPPxxxx/Beckhoff EPP2xxx/Beckhoff EPP2xxxEK1122/A_0079(EPP2816-0010-0017)
//     PlcTask Inputs/GVL_iXlinker.EtherCAT_Master_EPPxxxx.Beckhoff_EPP2xxx.Beckhoff_EPP2xxxEK1122.A_0079_EPP2816_0010_0017.DIG_Diag_Inputs_Channel_1.Diag_Input[0] <-> DIG Diag Inputs  Channel 1/Diag Input 1
//     PlcTask Inputs/GVL_iXlinker.EtherCAT_Master_EPPxxxx.Beckhoff_EPP2xxx.Beckhoff_EPP2xxxEK1122.A_0079_EPP2816_0010_0017.DIG_Diag_Inputs_Channel_1.Diag_Input[1] <-> DIG Diag Inputs  Channel 1/Diag Input 2
//     PlcTask Inputs/GVL_iXlinker.EtherCAT_Master_EPPxxxx.Beckhoff_EPP2xxx.Beckhoff_EPP2xxxEK1122.A_0079_EPP2816_0010_0017.DIG_Diag_Inputs_Channel_1.Diag_Input[2] <-> DIG Diag Inputs  Channel 1/Diag Input 3
//     PlcTask Inputs/GVL_iXlinker.EtherCAT_Master_EPPxxxx.Beckhoff_EPP2xxx.Beckhoff_EPP2xxxEK1122.A_0079_EPP2816_0010_0017.DIG_Diag_Inputs_Channel_1.Diag_Input[3] <-> DIG Diag Inputs  Channel 1/Diag Input 4
//     PlcTask Inputs/GVL_iXlinker.EtherCAT_Master_EPPxxxx.Beckhoff_EPP2xxx.Beckhoff_EPP2xxxEK1122.A_0079_EPP2816_0010_0017.DIG_Diag_Inputs_Channel_1.Diag_Input[4] <-> DIG Diag Inputs  Channel 1/Diag Input 5
//     PlcTask Inputs/GVL_iXlinker.EtherCAT_Master_EPPxxxx.Beckhoff_EPP2xxx.Beckhoff_EPP2xxxEK1122.A_0079_EPP2816_0010_0017.DIG_Diag_Inputs_Channel_1.Diag_Input[5] <-> DIG Diag Inputs  Channel 1/Diag Input 6
//     PlcTask Inputs/GVL_iXlinker.EtherCAT_Master_EPPxxxx.Beckhoff_EPP2xxx.Beckhoff_EPP2xxxEK1122.A_0079_EPP2816_0010_0017.DIG_Diag_Inputs_Channel_1.Diag_Input[6] <-> DIG Diag Inputs  Channel 1/Diag Input 7
//     PlcTask Inputs/GVL_iXlinker.EtherCAT_Master_EPPxxxx.Beckhoff_EPP2xxx.Beckhoff_EPP2xxxEK1122.A_0079_EPP2816_0010_0017.DIG_Diag_Inputs_Channel_1.Diag_Input[7] <-> DIG Diag Inputs  Channel 1/Diag Input 8
//     PlcTask Inputs/GVL_iXlinker.EtherCAT_Master_EPPxxxx.Beckhoff_EPP2xxx.Beckhoff_EPP2xxxEK1122.A_0079_EPP2816_0010_0017.DIG_Diag_Inputs_Channel_2.Diag_Input[0] <-> DIG Diag Inputs  Channel 2/Diag Input 1
//     PlcTask Inputs/GVL_iXlinker.EtherCAT_Master_EPPxxxx.Beckhoff_EPP2xxx.Beckhoff_EPP2xxxEK1122.A_0079_EPP2816_0010_0017.DIG_Diag_Inputs_Channel_2.Diag_Input[1] <-> DIG Diag Inputs  Channel 2/Diag Input 2
//     PlcTask Inputs/GVL_iXlinker.EtherCAT_Master_EPPxxxx.Beckhoff_EPP2xxx.Beckhoff_EPP2xxxEK1122.A_0079_EPP2816_0010_0017.DIG_Diag_Inputs_Channel_2.Diag_Input[2] <-> DIG Diag Inputs  Channel 2/Diag Input 3
//     PlcTask Inputs/GVL_iXlinker.EtherCAT_Master_EPPxxxx.Beckhoff_EPP2xxx.Beckhoff_EPP2xxxEK1122.A_0079_EPP2816_0010_0017.DIG_Diag_Inputs_Channel_2.Diag_Input[3] <-> DIG Diag Inputs  Channel 2/Diag Input 4
//     PlcTask Inputs/GVL_iXlinker.EtherCAT_Master_EPPxxxx.Beckhoff_EPP2xxx.Beckhoff_EPP2xxxEK1122.A_0079_EPP2816_0010_0017.DIG_Diag_Inputs_Channel_2.Diag_Input[4] <-> DIG Diag Inputs  Channel 2/Diag Input 5
//     PlcTask Inputs/GVL_iXlinker.EtherCAT_Master_EPPxxxx.Beckhoff_EPP2xxx.Beckhoff_EPP2xxxEK1122.A_0079_EPP2816_0010_0017.DIG_Diag_Inputs_Channel_2.Diag_Input[5] <-> DIG Diag Inputs  Channel 2/Diag Input 6
//     PlcTask Inputs/GVL_iXlinker.EtherCAT_Master_EPPxxxx.Beckhoff_EPP2xxx.Beckhoff_EPP2xxxEK1122.A_0079_EPP2816_0010_0017.DIG_Diag_Inputs_Channel_2.Diag_Input[6] <-> DIG Diag Inputs  Channel 2/Diag Input 7
//     PlcTask Inputs/GVL_iXlinker.EtherCAT_Master_EPPxxxx.Beckhoff_EPP2xxx.Beckhoff_EPP2xxxEK1122.A_0079_EPP2816_0010_0017.DIG_Diag_Inputs_Channel_2.Diag_Input[7] <-> DIG Diag Inputs  Channel 2/Diag Input 8
//     PlcTask Inputs/GVL_iXlinker.EtherCAT_Master_EPPxxxx.Beckhoff_EPP2xxx.Beckhoff_EPP2xxxEK1122.A_0079_EPP2816_0010_0017.DIG_Inputs_Device.Safe_state_active <-> DIG Inputs Device/Safe state active
//     PlcTask Inputs/GVL_iXlinker.EtherCAT_Master_EPPxxxx.Beckhoff_EPP2xxx.Beckhoff_EPP2xxxEK1122.A_0079_EPP2816_0010_0017.DIG_Inputs_Device.Error_channel[0] <-> DIG Inputs Device/Error channel 1
//     PlcTask Inputs/GVL_iXlinker.EtherCAT_Master_EPPxxxx.Beckhoff_EPP2xxx.Beckhoff_EPP2xxxEK1122.A_0079_EPP2816_0010_0017.DIG_Inputs_Device.Error_channel[1] <-> DIG Inputs Device/Error channel 2
//     PlcTask Inputs/GVL_iXlinker.EtherCAT_Master_EPPxxxx.Beckhoff_EPP2xxx.Beckhoff_EPP2xxxEK1122.A_0079_EPP2816_0010_0017.DIG_Inputs_Device.Sync_error <-> DIG Inputs Device/Sync error
//     PlcTask Inputs/GVL_iXlinker.EtherCAT_Master_EPPxxxx.Beckhoff_EPP2xxx.Beckhoff_EPP2xxxEK1122.A_0079_EPP2816_0010_0017.DIG_Inputs_Device.TxPDO_Toggle <-> DIG Inputs Device/TxPDO Toggle
//     PlcTask Outputs/GVL_iXlinker.EtherCAT_Master_EPPxxxx.Beckhoff_EPP2xxx.Beckhoff_EPP2xxxEK1122.A_0079_EPP2816_0010_0017.DIG_Outputs_Channel_1.Output[0] <-> DIG Outputs Channel 1/Output 1
//     PlcTask Outputs/GVL_iXlinker.EtherCAT_Master_EPPxxxx.Beckhoff_EPP2xxx.Beckhoff_EPP2xxxEK1122.A_0079_EPP2816_0010_0017.DIG_Outputs_Channel_1.Output[1] <-> DIG Outputs Channel 1/Output 2
//     PlcTask Outputs/GVL_iXlinker.EtherCAT_Master_EPPxxxx.Beckhoff_EPP2xxx.Beckhoff_EPP2xxxEK1122.A_0079_EPP2816_0010_0017.DIG_Outputs_Channel_1.Output[2] <-> DIG Outputs Channel 1/Output 3
//     PlcTask Outputs/GVL_iXlinker.EtherCAT_Master_EPPxxxx.Beckhoff_EPP2xxx.Beckhoff_EPP2xxxEK1122.A_0079_EPP2816_0010_0017.DIG_Outputs_Channel_1.Output[3] <-> DIG Outputs Channel 1/Output 4
//     PlcTask Outputs/GVL_iXlinker.EtherCAT_Master_EPPxxxx.Beckhoff_EPP2xxx.Beckhoff_EPP2xxxEK1122.A_0079_EPP2816_0010_0017.DIG_Outputs_Channel_1.Output[4] <-> DIG Outputs Channel 1/Output 5
//     PlcTask Outputs/GVL_iXlinker.EtherCAT_Master_EPPxxxx.Beckhoff_EPP2xxx.Beckhoff_EPP2xxxEK1122.A_0079_EPP2816_0010_0017.DIG_Outputs_Channel_1.Output[5] <-> DIG Outputs Channel 1/Output 6
//     PlcTask Outputs/GVL_iXlinker.EtherCAT_Master_EPPxxxx.Beckhoff_EPP2xxx.Beckhoff_EPP2xxxEK1122.A_0079_EPP2816_0010_0017.DIG_Outputs_Channel_1.Output[6] <-> DIG Outputs Channel 1/Output 7
//     PlcTask Outputs/GVL_iXlinker.EtherCAT_Master_EPPxxxx.Beckhoff_EPP2xxx.Beckhoff_EPP2xxxEK1122.A_0079_EPP2816_0010_0017.DIG_Outputs_Channel_1.Output[7] <-> DIG Outputs Channel 1/Output 8
//     PlcTask Outputs/GVL_iXlinker.EtherCAT_Master_EPPxxxx.Beckhoff_EPP2xxx.Beckhoff_EPP2xxxEK1122.A_0079_EPP2816_0010_0017.DIG_Outputs_Channel_2.Output[0] <-> DIG Outputs Channel 2/Output 1
//     PlcTask Outputs/GVL_iXlinker.EtherCAT_Master_EPPxxxx.Beckhoff_EPP2xxx.Beckhoff_EPP2xxxEK1122.A_0079_EPP2816_0010_0017.DIG_Outputs_Channel_2.Output[1] <-> DIG Outputs Channel 2/Output 2
//     PlcTask Outputs/GVL_iXlinker.EtherCAT_Master_EPPxxxx.Beckhoff_EPP2xxx.Beckhoff_EPP2xxxEK1122.A_0079_EPP2816_0010_0017.DIG_Outputs_Channel_2.Output[2] <-> DIG Outputs Channel 2/Output 3
//     PlcTask Outputs/GVL_iXlinker.EtherCAT_Master_EPPxxxx.Beckhoff_EPP2xxx.Beckhoff_EPP2xxxEK1122.A_0079_EPP2816_0010_0017.DIG_Outputs_Channel_2.Output[3] <-> DIG Outputs Channel 2/Output 4
//     PlcTask Outputs/GVL_iXlinker.EtherCAT_Master_EPPxxxx.Beckhoff_EPP2xxx.Beckhoff_EPP2xxxEK1122.A_0079_EPP2816_0010_0017.DIG_Outputs_Channel_2.Output[4] <-> DIG Outputs Channel 2/Output 5
//     PlcTask Outputs/GVL_iXlinker.EtherCAT_Master_EPPxxxx.Beckhoff_EPP2xxx.Beckhoff_EPP2xxxEK1122.A_0079_EPP2816_0010_0017.DIG_Outputs_Channel_2.Output[5] <-> DIG Outputs Channel 2/Output 6
//     PlcTask Outputs/GVL_iXlinker.EtherCAT_Master_EPPxxxx.Beckhoff_EPP2xxx.Beckhoff_EPP2xxxEK1122.A_0079_EPP2816_0010_0017.DIG_Outputs_Channel_2.Output[6] <-> DIG Outputs Channel 2/Output 7
//     PlcTask Outputs/GVL_iXlinker.EtherCAT_Master_EPPxxxx.Beckhoff_EPP2xxx.Beckhoff_EPP2xxxEK1122.A_0079_EPP2816_0010_0017.DIG_Outputs_Channel_2.Output[7] <-> DIG Outputs Channel 2/Output 8
//     PlcTask Outputs/GVL_iXlinker.EtherCAT_Master_EPPxxxx.Beckhoff_EPP2xxx.Beckhoff_EPP2xxxEK1122.A_0079_EPP2816_0010_0017.DIG_Outputs_Device.Set_safe_state <-> DIG Outputs Device/Set safe state
//     PlcTask Outputs/GVL_iXlinker.EtherCAT_Master_EPPxxxx.Beckhoff_EPP2xxx.Beckhoff_EPP2xxxEK1122.A_0079_EPP2816_0010_0017.DIG_Outputs_Device.Reset_outputs <-> DIG Outputs Device/Reset outputs
//     PlcTask Inputs/GVL_iXlinker.EtherCAT_Master_EPPxxxx.Beckhoff_EPP2xxx.Beckhoff_EPP2xxxEK1122.A_0079_EPP2816_0010_0017.WcState.WcState <-> WcState/WcState
//     PlcTask Inputs/GVL_iXlinker.EtherCAT_Master_EPPxxxx.Beckhoff_EPP2xxx.Beckhoff_EPP2xxxEK1122.A_0079_EPP2816_0010_0017.WcState.InputToggle <-> WcState/InputToggle
//     PlcTask Inputs/GVL_iXlinker.EtherCAT_Master_EPPxxxx.Beckhoff_EPP2xxx.Beckhoff_EPP2xxxEK1122.A_0079_EPP2816_0010_0017.InfoData.AdsAddr <-> InfoData/AdsAddr
//     PlcTask Inputs/GVL_iXlinker.EtherCAT_Master_EPPxxxx.Beckhoff_EPP2xxx.Beckhoff_EPP2xxxEK1122.A_0079_EPP2816_0010_0017.InfoData.State <-> InfoData/State
//   PLC/PLC Instance <-> EtherCAT Master EPPxxxx/Beckhoff EPP2xxx/Beckhoff EPP2xxxEK1122/A_0080(EPP2816-0010-0018)
//     PlcTask Inputs/GVL_iXlinker.EtherCAT_Master_EPPxxxx.Beckhoff_EPP2xxx.Beckhoff_EPP2xxxEK1122.A_0080_EPP2816_0010_0018.DIG_Diag_Inputs_Channel_1.Diag_Input[0] <-> DIG Diag Inputs  Channel 1/Diag Input 1
//     PlcTask Inputs/GVL_iXlinker.EtherCAT_Master_EPPxxxx.Beckhoff_EPP2xxx.Beckhoff_EPP2xxxEK1122.A_0080_EPP2816_0010_0018.DIG_Diag_Inputs_Channel_1.Diag_Input[1] <-> DIG Diag Inputs  Channel 1/Diag Input 2
//     PlcTask Inputs/GVL_iXlinker.EtherCAT_Master_EPPxxxx.Beckhoff_EPP2xxx.Beckhoff_EPP2xxxEK1122.A_0080_EPP2816_0010_0018.DIG_Diag_Inputs_Channel_1.Diag_Input[2] <-> DIG Diag Inputs  Channel 1/Diag Input 3
//     PlcTask Inputs/GVL_iXlinker.EtherCAT_Master_EPPxxxx.Beckhoff_EPP2xxx.Beckhoff_EPP2xxxEK1122.A_0080_EPP2816_0010_0018.DIG_Diag_Inputs_Channel_1.Diag_Input[3] <-> DIG Diag Inputs  Channel 1/Diag Input 4
//     PlcTask Inputs/GVL_iXlinker.EtherCAT_Master_EPPxxxx.Beckhoff_EPP2xxx.Beckhoff_EPP2xxxEK1122.A_0080_EPP2816_0010_0018.DIG_Diag_Inputs_Channel_1.Diag_Input[4] <-> DIG Diag Inputs  Channel 1/Diag Input 5
//     PlcTask Inputs/GVL_iXlinker.EtherCAT_Master_EPPxxxx.Beckhoff_EPP2xxx.Beckhoff_EPP2xxxEK1122.A_0080_EPP2816_0010_0018.DIG_Diag_Inputs_Channel_1.Diag_Input[5] <-> DIG Diag Inputs  Channel 1/Diag Input 6
//     PlcTask Inputs/GVL_iXlinker.EtherCAT_Master_EPPxxxx.Beckhoff_EPP2xxx.Beckhoff_EPP2xxxEK1122.A_0080_EPP2816_0010_0018.DIG_Diag_Inputs_Channel_1.Diag_Input[6] <-> DIG Diag Inputs  Channel 1/Diag Input 7
//     PlcTask Inputs/GVL_iXlinker.EtherCAT_Master_EPPxxxx.Beckhoff_EPP2xxx.Beckhoff_EPP2xxxEK1122.A_0080_EPP2816_0010_0018.DIG_Diag_Inputs_Channel_1.Diag_Input[7] <-> DIG Diag Inputs  Channel 1/Diag Input 8
//     PlcTask Inputs/GVL_iXlinker.EtherCAT_Master_EPPxxxx.Beckhoff_EPP2xxx.Beckhoff_EPP2xxxEK1122.A_0080_EPP2816_0010_0018.DIG_Diag_Inputs_Channel_2.Diag_Input[0] <-> DIG Diag Inputs  Channel 2/Diag Input 1
//     PlcTask Inputs/GVL_iXlinker.EtherCAT_Master_EPPxxxx.Beckhoff_EPP2xxx.Beckhoff_EPP2xxxEK1122.A_0080_EPP2816_0010_0018.DIG_Diag_Inputs_Channel_2.Diag_Input[1] <-> DIG Diag Inputs  Channel 2/Diag Input 2
//     PlcTask Inputs/GVL_iXlinker.EtherCAT_Master_EPPxxxx.Beckhoff_EPP2xxx.Beckhoff_EPP2xxxEK1122.A_0080_EPP2816_0010_0018.DIG_Diag_Inputs_Channel_2.Diag_Input[2] <-> DIG Diag Inputs  Channel 2/Diag Input 3
//     PlcTask Inputs/GVL_iXlinker.EtherCAT_Master_EPPxxxx.Beckhoff_EPP2xxx.Beckhoff_EPP2xxxEK1122.A_0080_EPP2816_0010_0018.DIG_Diag_Inputs_Channel_2.Diag_Input[3] <-> DIG Diag Inputs  Channel 2/Diag Input 4
//     PlcTask Inputs/GVL_iXlinker.EtherCAT_Master_EPPxxxx.Beckhoff_EPP2xxx.Beckhoff_EPP2xxxEK1122.A_0080_EPP2816_0010_0018.DIG_Diag_Inputs_Channel_2.Diag_Input[4] <-> DIG Diag Inputs  Channel 2/Diag Input 5
//     PlcTask Inputs/GVL_iXlinker.EtherCAT_Master_EPPxxxx.Beckhoff_EPP2xxx.Beckhoff_EPP2xxxEK1122.A_0080_EPP2816_0010_0018.DIG_Diag_Inputs_Channel_2.Diag_Input[5] <-> DIG Diag Inputs  Channel 2/Diag Input 6
//     PlcTask Inputs/GVL_iXlinker.EtherCAT_Master_EPPxxxx.Beckhoff_EPP2xxx.Beckhoff_EPP2xxxEK1122.A_0080_EPP2816_0010_0018.DIG_Diag_Inputs_Channel_2.Diag_Input[6] <-> DIG Diag Inputs  Channel 2/Diag Input 7
//     PlcTask Inputs/GVL_iXlinker.EtherCAT_Master_EPPxxxx.Beckhoff_EPP2xxx.Beckhoff_EPP2xxxEK1122.A_0080_EPP2816_0010_0018.DIG_Diag_Inputs_Channel_2.Diag_Input[7] <-> DIG Diag Inputs  Channel 2/Diag Input 8
//     PlcTask Inputs/GVL_iXlinker.EtherCAT_Master_EPPxxxx.Beckhoff_EPP2xxx.Beckhoff_EPP2xxxEK1122.A_0080_EPP2816_0010_0018.DIG_Inputs_Device.Safe_state_active <-> DIG Inputs Device/Safe state active
//     PlcTask Inputs/GVL_iXlinker.EtherCAT_Master_EPPxxxx.Beckhoff_EPP2xxx.Beckhoff_EPP2xxxEK1122.A_0080_EPP2816_0010_0018.DIG_Inputs_Device.Error_channel[0] <-> DIG Inputs Device/Error channel 1
//     PlcTask Inputs/GVL_iXlinker.EtherCAT_Master_EPPxxxx.Beckhoff_EPP2xxx.Beckhoff_EPP2xxxEK1122.A_0080_EPP2816_0010_0018.DIG_Inputs_Device.Error_channel[1] <-> DIG Inputs Device/Error channel 2
//     PlcTask Inputs/GVL_iXlinker.EtherCAT_Master_EPPxxxx.Beckhoff_EPP2xxx.Beckhoff_EPP2xxxEK1122.A_0080_EPP2816_0010_0018.DIG_Inputs_Device.Sync_error <-> DIG Inputs Device/Sync error
//     PlcTask Inputs/GVL_iXlinker.EtherCAT_Master_EPPxxxx.Beckhoff_EPP2xxx.Beckhoff_EPP2xxxEK1122.A_0080_EPP2816_0010_0018.DIG_Inputs_Device.TxPDO_Toggle <-> DIG Inputs Device/TxPDO Toggle
//     PlcTask Outputs/GVL_iXlinker.EtherCAT_Master_EPPxxxx.Beckhoff_EPP2xxx.Beckhoff_EPP2xxxEK1122.A_0080_EPP2816_0010_0018.DIG_Outputs_Channel_1.Output[0] <-> DIG Outputs Channel 1/Output 1
//     PlcTask Outputs/GVL_iXlinker.EtherCAT_Master_EPPxxxx.Beckhoff_EPP2xxx.Beckhoff_EPP2xxxEK1122.A_0080_EPP2816_0010_0018.DIG_Outputs_Channel_1.Output[1] <-> DIG Outputs Channel 1/Output 2
//     PlcTask Outputs/GVL_iXlinker.EtherCAT_Master_EPPxxxx.Beckhoff_EPP2xxx.Beckhoff_EPP2xxxEK1122.A_0080_EPP2816_0010_0018.DIG_Outputs_Channel_1.Output[2] <-> DIG Outputs Channel 1/Output 3
//     PlcTask Outputs/GVL_iXlinker.EtherCAT_Master_EPPxxxx.Beckhoff_EPP2xxx.Beckhoff_EPP2xxxEK1122.A_0080_EPP2816_0010_0018.DIG_Outputs_Channel_1.Output[3] <-> DIG Outputs Channel 1/Output 4
//     PlcTask Outputs/GVL_iXlinker.EtherCAT_Master_EPPxxxx.Beckhoff_EPP2xxx.Beckhoff_EPP2xxxEK1122.A_0080_EPP2816_0010_0018.DIG_Outputs_Channel_1.Output[4] <-> DIG Outputs Channel 1/Output 5
//     PlcTask Outputs/GVL_iXlinker.EtherCAT_Master_EPPxxxx.Beckhoff_EPP2xxx.Beckhoff_EPP2xxxEK1122.A_0080_EPP2816_0010_0018.DIG_Outputs_Channel_1.Output[5] <-> DIG Outputs Channel 1/Output 6
//     PlcTask Outputs/GVL_iXlinker.EtherCAT_Master_EPPxxxx.Beckhoff_EPP2xxx.Beckhoff_EPP2xxxEK1122.A_0080_EPP2816_0010_0018.DIG_Outputs_Channel_1.Output[6] <-> DIG Outputs Channel 1/Output 7
//     PlcTask Outputs/GVL_iXlinker.EtherCAT_Master_EPPxxxx.Beckhoff_EPP2xxx.Beckhoff_EPP2xxxEK1122.A_0080_EPP2816_0010_0018.DIG_Outputs_Channel_1.Output[7] <-> DIG Outputs Channel 1/Output 8
//     PlcTask Outputs/GVL_iXlinker.EtherCAT_Master_EPPxxxx.Beckhoff_EPP2xxx.Beckhoff_EPP2xxxEK1122.A_0080_EPP2816_0010_0018.DIG_Outputs_Channel_2.Output[0] <-> DIG Outputs Channel 2/Output 1
//     PlcTask Outputs/GVL_iXlinker.EtherCAT_Master_EPPxxxx.Beckhoff_EPP2xxx.Beckhoff_EPP2xxxEK1122.A_0080_EPP2816_0010_0018.DIG_Outputs_Channel_2.Output[1] <-> DIG Outputs Channel 2/Output 2
//     PlcTask Outputs/GVL_iXlinker.EtherCAT_Master_EPPxxxx.Beckhoff_EPP2xxx.Beckhoff_EPP2xxxEK1122.A_0080_EPP2816_0010_0018.DIG_Outputs_Channel_2.Output[2] <-> DIG Outputs Channel 2/Output 3
//     PlcTask Outputs/GVL_iXlinker.EtherCAT_Master_EPPxxxx.Beckhoff_EPP2xxx.Beckhoff_EPP2xxxEK1122.A_0080_EPP2816_0010_0018.DIG_Outputs_Channel_2.Output[3] <-> DIG Outputs Channel 2/Output 4
//     PlcTask Outputs/GVL_iXlinker.EtherCAT_Master_EPPxxxx.Beckhoff_EPP2xxx.Beckhoff_EPP2xxxEK1122.A_0080_EPP2816_0010_0018.DIG_Outputs_Channel_2.Output[4] <-> DIG Outputs Channel 2/Output 5
//     PlcTask Outputs/GVL_iXlinker.EtherCAT_Master_EPPxxxx.Beckhoff_EPP2xxx.Beckhoff_EPP2xxxEK1122.A_0080_EPP2816_0010_0018.DIG_Outputs_Channel_2.Output[5] <-> DIG Outputs Channel 2/Output 6
//     PlcTask Outputs/GVL_iXlinker.EtherCAT_Master_EPPxxxx.Beckhoff_EPP2xxx.Beckhoff_EPP2xxxEK1122.A_0080_EPP2816_0010_0018.DIG_Outputs_Channel_2.Output[6] <-> DIG Outputs Channel 2/Output 7
//     PlcTask Outputs/GVL_iXlinker.EtherCAT_Master_EPPxxxx.Beckhoff_EPP2xxx.Beckhoff_EPP2xxxEK1122.A_0080_EPP2816_0010_0018.DIG_Outputs_Channel_2.Output[7] <-> DIG Outputs Channel 2/Output 8
//     PlcTask Outputs/GVL_iXlinker.EtherCAT_Master_EPPxxxx.Beckhoff_EPP2xxx.Beckhoff_EPP2xxxEK1122.A_0080_EPP2816_0010_0018.DIG_Outputs_Device.Set_safe_state <-> DIG Outputs Device/Set safe state
//     PlcTask Outputs/GVL_iXlinker.EtherCAT_Master_EPPxxxx.Beckhoff_EPP2xxx.Beckhoff_EPP2xxxEK1122.A_0080_EPP2816_0010_0018.DIG_Outputs_Device.Reset_outputs <-> DIG Outputs Device/Reset outputs
//     PlcTask Inputs/GVL_iXlinker.EtherCAT_Master_EPPxxxx.Beckhoff_EPP2xxx.Beckhoff_EPP2xxxEK1122.A_0080_EPP2816_0010_0018.WcState.WcState <-> WcState/WcState
//     PlcTask Inputs/GVL_iXlinker.EtherCAT_Master_EPPxxxx.Beckhoff_EPP2xxx.Beckhoff_EPP2xxxEK1122.A_0080_EPP2816_0010_0018.WcState.InputToggle <-> WcState/InputToggle
//     PlcTask Inputs/GVL_iXlinker.EtherCAT_Master_EPPxxxx.Beckhoff_EPP2xxx.Beckhoff_EPP2xxxEK1122.A_0080_EPP2816_0010_0018.InfoData.AdsAddr <-> InfoData/AdsAddr
//     PlcTask Inputs/GVL_iXlinker.EtherCAT_Master_EPPxxxx.Beckhoff_EPP2xxx.Beckhoff_EPP2xxxEK1122.A_0080_EPP2816_0010_0018.InfoData.State <-> InfoData/State
//   PLC/PLC Instance <-> EtherCAT Master EPPxxxx/Beckhoff EPP2xxx/Beckhoff EPP2xxxEK1122/A_0081(EPP2817-0008-0016)
//     PlcTask Inputs/GVL_iXlinker.EtherCAT_Master_EPPxxxx.Beckhoff_EPP2xxx.Beckhoff_EPP2xxxEK1122.A_0081_EPP2817_0008_0016.DIG_Diag_Inputs_Channel_1.Diag_Input[0] <-> DIG Diag Inputs Channel 1/Diag Input 1
//     PlcTask Inputs/GVL_iXlinker.EtherCAT_Master_EPPxxxx.Beckhoff_EPP2xxx.Beckhoff_EPP2xxxEK1122.A_0081_EPP2817_0008_0016.DIG_Diag_Inputs_Channel_1.Diag_Input[1] <-> DIG Diag Inputs Channel 1/Diag Input 2
//     PlcTask Inputs/GVL_iXlinker.EtherCAT_Master_EPPxxxx.Beckhoff_EPP2xxx.Beckhoff_EPP2xxxEK1122.A_0081_EPP2817_0008_0016.DIG_Diag_Inputs_Channel_1.Diag_Input[2] <-> DIG Diag Inputs Channel 1/Diag Input 3
//     PlcTask Inputs/GVL_iXlinker.EtherCAT_Master_EPPxxxx.Beckhoff_EPP2xxx.Beckhoff_EPP2xxxEK1122.A_0081_EPP2817_0008_0016.DIG_Diag_Inputs_Channel_1.Diag_Input[3] <-> DIG Diag Inputs Channel 1/Diag Input 4
//     PlcTask Inputs/GVL_iXlinker.EtherCAT_Master_EPPxxxx.Beckhoff_EPP2xxx.Beckhoff_EPP2xxxEK1122.A_0081_EPP2817_0008_0016.DIG_Diag_Inputs_Channel_1.Diag_Input[4] <-> DIG Diag Inputs Channel 1/Diag Input 5
//     PlcTask Inputs/GVL_iXlinker.EtherCAT_Master_EPPxxxx.Beckhoff_EPP2xxx.Beckhoff_EPP2xxxEK1122.A_0081_EPP2817_0008_0016.DIG_Diag_Inputs_Channel_1.Diag_Input[5] <-> DIG Diag Inputs Channel 1/Diag Input 6
//     PlcTask Inputs/GVL_iXlinker.EtherCAT_Master_EPPxxxx.Beckhoff_EPP2xxx.Beckhoff_EPP2xxxEK1122.A_0081_EPP2817_0008_0016.DIG_Diag_Inputs_Channel_1.Diag_Input[6] <-> DIG Diag Inputs Channel 1/Diag Input 7
//     PlcTask Inputs/GVL_iXlinker.EtherCAT_Master_EPPxxxx.Beckhoff_EPP2xxx.Beckhoff_EPP2xxxEK1122.A_0081_EPP2817_0008_0016.DIG_Diag_Inputs_Channel_1.Diag_Input[7] <-> DIG Diag Inputs Channel 1/Diag Input 8
//     PlcTask Inputs/GVL_iXlinker.EtherCAT_Master_EPPxxxx.Beckhoff_EPP2xxx.Beckhoff_EPP2xxxEK1122.A_0081_EPP2817_0008_0016.DIG_Diag_Inputs_Channel_2.Diag_Input[0] <-> DIG Diag Inputs Channel 2/Diag Input 1
//     PlcTask Inputs/GVL_iXlinker.EtherCAT_Master_EPPxxxx.Beckhoff_EPP2xxx.Beckhoff_EPP2xxxEK1122.A_0081_EPP2817_0008_0016.DIG_Diag_Inputs_Channel_2.Diag_Input[1] <-> DIG Diag Inputs Channel 2/Diag Input 2
//     PlcTask Inputs/GVL_iXlinker.EtherCAT_Master_EPPxxxx.Beckhoff_EPP2xxx.Beckhoff_EPP2xxxEK1122.A_0081_EPP2817_0008_0016.DIG_Diag_Inputs_Channel_2.Diag_Input[2] <-> DIG Diag Inputs Channel 2/Diag Input 3
//     PlcTask Inputs/GVL_iXlinker.EtherCAT_Master_EPPxxxx.Beckhoff_EPP2xxx.Beckhoff_EPP2xxxEK1122.A_0081_EPP2817_0008_0016.DIG_Diag_Inputs_Channel_2.Diag_Input[3] <-> DIG Diag Inputs Channel 2/Diag Input 4
//     PlcTask Inputs/GVL_iXlinker.EtherCAT_Master_EPPxxxx.Beckhoff_EPP2xxx.Beckhoff_EPP2xxxEK1122.A_0081_EPP2817_0008_0016.DIG_Diag_Inputs_Channel_2.Diag_Input[4] <-> DIG Diag Inputs Channel 2/Diag Input 5
//     PlcTask Inputs/GVL_iXlinker.EtherCAT_Master_EPPxxxx.Beckhoff_EPP2xxx.Beckhoff_EPP2xxxEK1122.A_0081_EPP2817_0008_0016.DIG_Diag_Inputs_Channel_2.Diag_Input[5] <-> DIG Diag Inputs Channel 2/Diag Input 6
//     PlcTask Inputs/GVL_iXlinker.EtherCAT_Master_EPPxxxx.Beckhoff_EPP2xxx.Beckhoff_EPP2xxxEK1122.A_0081_EPP2817_0008_0016.DIG_Diag_Inputs_Channel_2.Diag_Input[6] <-> DIG Diag Inputs Channel 2/Diag Input 7
//     PlcTask Inputs/GVL_iXlinker.EtherCAT_Master_EPPxxxx.Beckhoff_EPP2xxx.Beckhoff_EPP2xxxEK1122.A_0081_EPP2817_0008_0016.DIG_Diag_Inputs_Channel_2.Diag_Input[7] <-> DIG Diag Inputs Channel 2/Diag Input 8
//     PlcTask Inputs/GVL_iXlinker.EtherCAT_Master_EPPxxxx.Beckhoff_EPP2xxx.Beckhoff_EPP2xxxEK1122.A_0081_EPP2817_0008_0016.DIG_Diag_Inputs_Channel_3.Diag_Input[0] <-> DIG Diag Inputs Channel 3/Diag Input 1
//     PlcTask Inputs/GVL_iXlinker.EtherCAT_Master_EPPxxxx.Beckhoff_EPP2xxx.Beckhoff_EPP2xxxEK1122.A_0081_EPP2817_0008_0016.DIG_Diag_Inputs_Channel_3.Diag_Input[1] <-> DIG Diag Inputs Channel 3/Diag Input 2
//     PlcTask Inputs/GVL_iXlinker.EtherCAT_Master_EPPxxxx.Beckhoff_EPP2xxx.Beckhoff_EPP2xxxEK1122.A_0081_EPP2817_0008_0016.DIG_Diag_Inputs_Channel_3.Diag_Input[2] <-> DIG Diag Inputs Channel 3/Diag Input 3
//     PlcTask Inputs/GVL_iXlinker.EtherCAT_Master_EPPxxxx.Beckhoff_EPP2xxx.Beckhoff_EPP2xxxEK1122.A_0081_EPP2817_0008_0016.DIG_Diag_Inputs_Channel_3.Diag_Input[3] <-> DIG Diag Inputs Channel 3/Diag Input 4
//     PlcTask Inputs/GVL_iXlinker.EtherCAT_Master_EPPxxxx.Beckhoff_EPP2xxx.Beckhoff_EPP2xxxEK1122.A_0081_EPP2817_0008_0016.DIG_Diag_Inputs_Channel_3.Diag_Input[4] <-> DIG Diag Inputs Channel 3/Diag Input 5
//     PlcTask Inputs/GVL_iXlinker.EtherCAT_Master_EPPxxxx.Beckhoff_EPP2xxx.Beckhoff_EPP2xxxEK1122.A_0081_EPP2817_0008_0016.DIG_Diag_Inputs_Channel_3.Diag_Input[5] <-> DIG Diag Inputs Channel 3/Diag Input 6
//     PlcTask Inputs/GVL_iXlinker.EtherCAT_Master_EPPxxxx.Beckhoff_EPP2xxx.Beckhoff_EPP2xxxEK1122.A_0081_EPP2817_0008_0016.DIG_Diag_Inputs_Channel_3.Diag_Input[6] <-> DIG Diag Inputs Channel 3/Diag Input 7
//     PlcTask Inputs/GVL_iXlinker.EtherCAT_Master_EPPxxxx.Beckhoff_EPP2xxx.Beckhoff_EPP2xxxEK1122.A_0081_EPP2817_0008_0016.DIG_Diag_Inputs_Channel_3.Diag_Input[7] <-> DIG Diag Inputs Channel 3/Diag Input 8
//     PlcTask Inputs/GVL_iXlinker.EtherCAT_Master_EPPxxxx.Beckhoff_EPP2xxx.Beckhoff_EPP2xxxEK1122.A_0081_EPP2817_0008_0016.DIG_Inputs_Device.Safe_state_active <-> DIG Inputs Device/Safe state active
//     PlcTask Inputs/GVL_iXlinker.EtherCAT_Master_EPPxxxx.Beckhoff_EPP2xxx.Beckhoff_EPP2xxxEK1122.A_0081_EPP2817_0008_0016.DIG_Inputs_Device.Error_channel[0] <-> DIG Inputs Device/Error channel 1
//     PlcTask Inputs/GVL_iXlinker.EtherCAT_Master_EPPxxxx.Beckhoff_EPP2xxx.Beckhoff_EPP2xxxEK1122.A_0081_EPP2817_0008_0016.DIG_Inputs_Device.Error_channel[1] <-> DIG Inputs Device/Error channel 2
//     PlcTask Inputs/GVL_iXlinker.EtherCAT_Master_EPPxxxx.Beckhoff_EPP2xxx.Beckhoff_EPP2xxxEK1122.A_0081_EPP2817_0008_0016.DIG_Inputs_Device.Error_channel[2] <-> DIG Inputs Device/Error channel 3
//     PlcTask Inputs/GVL_iXlinker.EtherCAT_Master_EPPxxxx.Beckhoff_EPP2xxx.Beckhoff_EPP2xxxEK1122.A_0081_EPP2817_0008_0016.DIG_Inputs_Device.Us_Undervoltage <-> DIG Inputs Device/Us Undervoltage
//     PlcTask Inputs/GVL_iXlinker.EtherCAT_Master_EPPxxxx.Beckhoff_EPP2xxx.Beckhoff_EPP2xxxEK1122.A_0081_EPP2817_0008_0016.DIG_Inputs_Device.Up_Undervoltage <-> DIG Inputs Device/Up Undervoltage
//     PlcTask Inputs/GVL_iXlinker.EtherCAT_Master_EPPxxxx.Beckhoff_EPP2xxx.Beckhoff_EPP2xxxEK1122.A_0081_EPP2817_0008_0016.DIG_Inputs_Device.Sync_error <-> DIG Inputs Device/Sync error
//     PlcTask Inputs/GVL_iXlinker.EtherCAT_Master_EPPxxxx.Beckhoff_EPP2xxx.Beckhoff_EPP2xxxEK1122.A_0081_EPP2817_0008_0016.DIG_Inputs_Device.TxPDO_Toggle <-> DIG Inputs Device/TxPDO Toggle
//     PlcTask Outputs/GVL_iXlinker.EtherCAT_Master_EPPxxxx.Beckhoff_EPP2xxx.Beckhoff_EPP2xxxEK1122.A_0081_EPP2817_0008_0016.DIG_Output_Channel_1.Output[0] <-> DIG Output Channel 1/Output 1
//     PlcTask Outputs/GVL_iXlinker.EtherCAT_Master_EPPxxxx.Beckhoff_EPP2xxx.Beckhoff_EPP2xxxEK1122.A_0081_EPP2817_0008_0016.DIG_Output_Channel_1.Output[1] <-> DIG Output Channel 1/Output 2
//     PlcTask Outputs/GVL_iXlinker.EtherCAT_Master_EPPxxxx.Beckhoff_EPP2xxx.Beckhoff_EPP2xxxEK1122.A_0081_EPP2817_0008_0016.DIG_Output_Channel_1.Output[2] <-> DIG Output Channel 1/Output 3
//     PlcTask Outputs/GVL_iXlinker.EtherCAT_Master_EPPxxxx.Beckhoff_EPP2xxx.Beckhoff_EPP2xxxEK1122.A_0081_EPP2817_0008_0016.DIG_Output_Channel_1.Output[3] <-> DIG Output Channel 1/Output 4
//     PlcTask Outputs/GVL_iXlinker.EtherCAT_Master_EPPxxxx.Beckhoff_EPP2xxx.Beckhoff_EPP2xxxEK1122.A_0081_EPP2817_0008_0016.DIG_Output_Channel_1.Output[4] <-> DIG Output Channel 1/Output 5
//     PlcTask Outputs/GVL_iXlinker.EtherCAT_Master_EPPxxxx.Beckhoff_EPP2xxx.Beckhoff_EPP2xxxEK1122.A_0081_EPP2817_0008_0016.DIG_Output_Channel_1.Output[5] <-> DIG Output Channel 1/Output 6
//     PlcTask Outputs/GVL_iXlinker.EtherCAT_Master_EPPxxxx.Beckhoff_EPP2xxx.Beckhoff_EPP2xxxEK1122.A_0081_EPP2817_0008_0016.DIG_Output_Channel_1.Output[6] <-> DIG Output Channel 1/Output 7
//     PlcTask Outputs/GVL_iXlinker.EtherCAT_Master_EPPxxxx.Beckhoff_EPP2xxx.Beckhoff_EPP2xxxEK1122.A_0081_EPP2817_0008_0016.DIG_Output_Channel_1.Output[7] <-> DIG Output Channel 1/Output 8
//     PlcTask Outputs/GVL_iXlinker.EtherCAT_Master_EPPxxxx.Beckhoff_EPP2xxx.Beckhoff_EPP2xxxEK1122.A_0081_EPP2817_0008_0016.DIG_Output_Channel_2.Output[0] <-> DIG Output Channel 2/Output 1
//     PlcTask Outputs/GVL_iXlinker.EtherCAT_Master_EPPxxxx.Beckhoff_EPP2xxx.Beckhoff_EPP2xxxEK1122.A_0081_EPP2817_0008_0016.DIG_Output_Channel_2.Output[1] <-> DIG Output Channel 2/Output 2
//     PlcTask Outputs/GVL_iXlinker.EtherCAT_Master_EPPxxxx.Beckhoff_EPP2xxx.Beckhoff_EPP2xxxEK1122.A_0081_EPP2817_0008_0016.DIG_Output_Channel_2.Output[2] <-> DIG Output Channel 2/Output 3
//     PlcTask Outputs/GVL_iXlinker.EtherCAT_Master_EPPxxxx.Beckhoff_EPP2xxx.Beckhoff_EPP2xxxEK1122.A_0081_EPP2817_0008_0016.DIG_Output_Channel_2.Output[3] <-> DIG Output Channel 2/Output 4
//     PlcTask Outputs/GVL_iXlinker.EtherCAT_Master_EPPxxxx.Beckhoff_EPP2xxx.Beckhoff_EPP2xxxEK1122.A_0081_EPP2817_0008_0016.DIG_Output_Channel_2.Output[4] <-> DIG Output Channel 2/Output 5
//     PlcTask Outputs/GVL_iXlinker.EtherCAT_Master_EPPxxxx.Beckhoff_EPP2xxx.Beckhoff_EPP2xxxEK1122.A_0081_EPP2817_0008_0016.DIG_Output_Channel_2.Output[5] <-> DIG Output Channel 2/Output 6
//     PlcTask Outputs/GVL_iXlinker.EtherCAT_Master_EPPxxxx.Beckhoff_EPP2xxx.Beckhoff_EPP2xxxEK1122.A_0081_EPP2817_0008_0016.DIG_Output_Channel_2.Output[6] <-> DIG Output Channel 2/Output 7
//     PlcTask Outputs/GVL_iXlinker.EtherCAT_Master_EPPxxxx.Beckhoff_EPP2xxx.Beckhoff_EPP2xxxEK1122.A_0081_EPP2817_0008_0016.DIG_Output_Channel_2.Output[7] <-> DIG Output Channel 2/Output 8
//     PlcTask Outputs/GVL_iXlinker.EtherCAT_Master_EPPxxxx.Beckhoff_EPP2xxx.Beckhoff_EPP2xxxEK1122.A_0081_EPP2817_0008_0016.DIG_Output_Channel_3.Output[0] <-> DIG Output Channel 3/Output 1
//     PlcTask Outputs/GVL_iXlinker.EtherCAT_Master_EPPxxxx.Beckhoff_EPP2xxx.Beckhoff_EPP2xxxEK1122.A_0081_EPP2817_0008_0016.DIG_Output_Channel_3.Output[1] <-> DIG Output Channel 3/Output 2
//     PlcTask Outputs/GVL_iXlinker.EtherCAT_Master_EPPxxxx.Beckhoff_EPP2xxx.Beckhoff_EPP2xxxEK1122.A_0081_EPP2817_0008_0016.DIG_Output_Channel_3.Output[2] <-> DIG Output Channel 3/Output 3
//     PlcTask Outputs/GVL_iXlinker.EtherCAT_Master_EPPxxxx.Beckhoff_EPP2xxx.Beckhoff_EPP2xxxEK1122.A_0081_EPP2817_0008_0016.DIG_Output_Channel_3.Output[3] <-> DIG Output Channel 3/Output 4
//     PlcTask Outputs/GVL_iXlinker.EtherCAT_Master_EPPxxxx.Beckhoff_EPP2xxx.Beckhoff_EPP2xxxEK1122.A_0081_EPP2817_0008_0016.DIG_Output_Channel_3.Output[4] <-> DIG Output Channel 3/Output 5
//     PlcTask Outputs/GVL_iXlinker.EtherCAT_Master_EPPxxxx.Beckhoff_EPP2xxx.Beckhoff_EPP2xxxEK1122.A_0081_EPP2817_0008_0016.DIG_Output_Channel_3.Output[5] <-> DIG Output Channel 3/Output 6
//     PlcTask Outputs/GVL_iXlinker.EtherCAT_Master_EPPxxxx.Beckhoff_EPP2xxx.Beckhoff_EPP2xxxEK1122.A_0081_EPP2817_0008_0016.DIG_Output_Channel_3.Output[6] <-> DIG Output Channel 3/Output 7
//     PlcTask Outputs/GVL_iXlinker.EtherCAT_Master_EPPxxxx.Beckhoff_EPP2xxx.Beckhoff_EPP2xxxEK1122.A_0081_EPP2817_0008_0016.DIG_Output_Channel_3.Output[7] <-> DIG Output Channel 3/Output 8
//     PlcTask Outputs/GVL_iXlinker.EtherCAT_Master_EPPxxxx.Beckhoff_EPP2xxx.Beckhoff_EPP2xxxEK1122.A_0081_EPP2817_0008_0016.DIG_Outputs_Device.Set_safe_state <-> DIG Outputs Device/Set safe state
//     PlcTask Outputs/GVL_iXlinker.EtherCAT_Master_EPPxxxx.Beckhoff_EPP2xxx.Beckhoff_EPP2xxxEK1122.A_0081_EPP2817_0008_0016.DIG_Outputs_Device.Reset_outputs <-> DIG Outputs Device/Reset outputs
//     PlcTask Inputs/GVL_iXlinker.EtherCAT_Master_EPPxxxx.Beckhoff_EPP2xxx.Beckhoff_EPP2xxxEK1122.A_0081_EPP2817_0008_0016.WcState.WcState <-> WcState/WcState
//     PlcTask Inputs/GVL_iXlinker.EtherCAT_Master_EPPxxxx.Beckhoff_EPP2xxx.Beckhoff_EPP2xxxEK1122.A_0081_EPP2817_0008_0016.WcState.InputToggle <-> WcState/InputToggle
//     PlcTask Inputs/GVL_iXlinker.EtherCAT_Master_EPPxxxx.Beckhoff_EPP2xxx.Beckhoff_EPP2xxxEK1122.A_0081_EPP2817_0008_0016.InfoData.AdsAddr <-> InfoData/AdsAddr
//     PlcTask Inputs/GVL_iXlinker.EtherCAT_Master_EPPxxxx.Beckhoff_EPP2xxx.Beckhoff_EPP2xxxEK1122.A_0081_EPP2817_0008_0016.InfoData.State <-> InfoData/State
//   PLC/PLC Instance <-> EtherCAT Master EPPxxxx/Beckhoff EPP2xxx/Beckhoff EPP2xxxEK1122/A_0082(EPP2817-0008-0017)
//     PlcTask Inputs/GVL_iXlinker.EtherCAT_Master_EPPxxxx.Beckhoff_EPP2xxx.Beckhoff_EPP2xxxEK1122.A_0082_EPP2817_0008_0017.DIG_Diag_Inputs_Channel_1.Diag_Input[0] <-> DIG Diag Inputs Channel 1/Diag Input 1
//     PlcTask Inputs/GVL_iXlinker.EtherCAT_Master_EPPxxxx.Beckhoff_EPP2xxx.Beckhoff_EPP2xxxEK1122.A_0082_EPP2817_0008_0017.DIG_Diag_Inputs_Channel_1.Diag_Input[1] <-> DIG Diag Inputs Channel 1/Diag Input 2
//     PlcTask Inputs/GVL_iXlinker.EtherCAT_Master_EPPxxxx.Beckhoff_EPP2xxx.Beckhoff_EPP2xxxEK1122.A_0082_EPP2817_0008_0017.DIG_Diag_Inputs_Channel_1.Diag_Input[2] <-> DIG Diag Inputs Channel 1/Diag Input 3
//     PlcTask Inputs/GVL_iXlinker.EtherCAT_Master_EPPxxxx.Beckhoff_EPP2xxx.Beckhoff_EPP2xxxEK1122.A_0082_EPP2817_0008_0017.DIG_Diag_Inputs_Channel_1.Diag_Input[3] <-> DIG Diag Inputs Channel 1/Diag Input 4
//     PlcTask Inputs/GVL_iXlinker.EtherCAT_Master_EPPxxxx.Beckhoff_EPP2xxx.Beckhoff_EPP2xxxEK1122.A_0082_EPP2817_0008_0017.DIG_Diag_Inputs_Channel_1.Diag_Input[4] <-> DIG Diag Inputs Channel 1/Diag Input 5
//     PlcTask Inputs/GVL_iXlinker.EtherCAT_Master_EPPxxxx.Beckhoff_EPP2xxx.Beckhoff_EPP2xxxEK1122.A_0082_EPP2817_0008_0017.DIG_Diag_Inputs_Channel_1.Diag_Input[5] <-> DIG Diag Inputs Channel 1/Diag Input 6
//     PlcTask Inputs/GVL_iXlinker.EtherCAT_Master_EPPxxxx.Beckhoff_EPP2xxx.Beckhoff_EPP2xxxEK1122.A_0082_EPP2817_0008_0017.DIG_Diag_Inputs_Channel_1.Diag_Input[6] <-> DIG Diag Inputs Channel 1/Diag Input 7
//     PlcTask Inputs/GVL_iXlinker.EtherCAT_Master_EPPxxxx.Beckhoff_EPP2xxx.Beckhoff_EPP2xxxEK1122.A_0082_EPP2817_0008_0017.DIG_Diag_Inputs_Channel_1.Diag_Input[7] <-> DIG Diag Inputs Channel 1/Diag Input 8
//     PlcTask Inputs/GVL_iXlinker.EtherCAT_Master_EPPxxxx.Beckhoff_EPP2xxx.Beckhoff_EPP2xxxEK1122.A_0082_EPP2817_0008_0017.DIG_Diag_Inputs_Channel_2.Diag_Input[0] <-> DIG Diag Inputs Channel 2/Diag Input 1
//     PlcTask Inputs/GVL_iXlinker.EtherCAT_Master_EPPxxxx.Beckhoff_EPP2xxx.Beckhoff_EPP2xxxEK1122.A_0082_EPP2817_0008_0017.DIG_Diag_Inputs_Channel_2.Diag_Input[1] <-> DIG Diag Inputs Channel 2/Diag Input 2
//     PlcTask Inputs/GVL_iXlinker.EtherCAT_Master_EPPxxxx.Beckhoff_EPP2xxx.Beckhoff_EPP2xxxEK1122.A_0082_EPP2817_0008_0017.DIG_Diag_Inputs_Channel_2.Diag_Input[2] <-> DIG Diag Inputs Channel 2/Diag Input 3
//     PlcTask Inputs/GVL_iXlinker.EtherCAT_Master_EPPxxxx.Beckhoff_EPP2xxx.Beckhoff_EPP2xxxEK1122.A_0082_EPP2817_0008_0017.DIG_Diag_Inputs_Channel_2.Diag_Input[3] <-> DIG Diag Inputs Channel 2/Diag Input 4
//     PlcTask Inputs/GVL_iXlinker.EtherCAT_Master_EPPxxxx.Beckhoff_EPP2xxx.Beckhoff_EPP2xxxEK1122.A_0082_EPP2817_0008_0017.DIG_Diag_Inputs_Channel_2.Diag_Input[4] <-> DIG Diag Inputs Channel 2/Diag Input 5
//     PlcTask Inputs/GVL_iXlinker.EtherCAT_Master_EPPxxxx.Beckhoff_EPP2xxx.Beckhoff_EPP2xxxEK1122.A_0082_EPP2817_0008_0017.DIG_Diag_Inputs_Channel_2.Diag_Input[5] <-> DIG Diag Inputs Channel 2/Diag Input 6
//     PlcTask Inputs/GVL_iXlinker.EtherCAT_Master_EPPxxxx.Beckhoff_EPP2xxx.Beckhoff_EPP2xxxEK1122.A_0082_EPP2817_0008_0017.DIG_Diag_Inputs_Channel_2.Diag_Input[6] <-> DIG Diag Inputs Channel 2/Diag Input 7
//     PlcTask Inputs/GVL_iXlinker.EtherCAT_Master_EPPxxxx.Beckhoff_EPP2xxx.Beckhoff_EPP2xxxEK1122.A_0082_EPP2817_0008_0017.DIG_Diag_Inputs_Channel_2.Diag_Input[7] <-> DIG Diag Inputs Channel 2/Diag Input 8
//     PlcTask Inputs/GVL_iXlinker.EtherCAT_Master_EPPxxxx.Beckhoff_EPP2xxx.Beckhoff_EPP2xxxEK1122.A_0082_EPP2817_0008_0017.DIG_Diag_Inputs_Channel_3.Diag_Input[0] <-> DIG Diag Inputs Channel 3/Diag Input 1
//     PlcTask Inputs/GVL_iXlinker.EtherCAT_Master_EPPxxxx.Beckhoff_EPP2xxx.Beckhoff_EPP2xxxEK1122.A_0082_EPP2817_0008_0017.DIG_Diag_Inputs_Channel_3.Diag_Input[1] <-> DIG Diag Inputs Channel 3/Diag Input 2
//     PlcTask Inputs/GVL_iXlinker.EtherCAT_Master_EPPxxxx.Beckhoff_EPP2xxx.Beckhoff_EPP2xxxEK1122.A_0082_EPP2817_0008_0017.DIG_Diag_Inputs_Channel_3.Diag_Input[2] <-> DIG Diag Inputs Channel 3/Diag Input 3
//     PlcTask Inputs/GVL_iXlinker.EtherCAT_Master_EPPxxxx.Beckhoff_EPP2xxx.Beckhoff_EPP2xxxEK1122.A_0082_EPP2817_0008_0017.DIG_Diag_Inputs_Channel_3.Diag_Input[3] <-> DIG Diag Inputs Channel 3/Diag Input 4
//     PlcTask Inputs/GVL_iXlinker.EtherCAT_Master_EPPxxxx.Beckhoff_EPP2xxx.Beckhoff_EPP2xxxEK1122.A_0082_EPP2817_0008_0017.DIG_Diag_Inputs_Channel_3.Diag_Input[4] <-> DIG Diag Inputs Channel 3/Diag Input 5
//     PlcTask Inputs/GVL_iXlinker.EtherCAT_Master_EPPxxxx.Beckhoff_EPP2xxx.Beckhoff_EPP2xxxEK1122.A_0082_EPP2817_0008_0017.DIG_Diag_Inputs_Channel_3.Diag_Input[5] <-> DIG Diag Inputs Channel 3/Diag Input 6
//     PlcTask Inputs/GVL_iXlinker.EtherCAT_Master_EPPxxxx.Beckhoff_EPP2xxx.Beckhoff_EPP2xxxEK1122.A_0082_EPP2817_0008_0017.DIG_Diag_Inputs_Channel_3.Diag_Input[6] <-> DIG Diag Inputs Channel 3/Diag Input 7
//     PlcTask Inputs/GVL_iXlinker.EtherCAT_Master_EPPxxxx.Beckhoff_EPP2xxx.Beckhoff_EPP2xxxEK1122.A_0082_EPP2817_0008_0017.DIG_Diag_Inputs_Channel_3.Diag_Input[7] <-> DIG Diag Inputs Channel 3/Diag Input 8
//     PlcTask Inputs/GVL_iXlinker.EtherCAT_Master_EPPxxxx.Beckhoff_EPP2xxx.Beckhoff_EPP2xxxEK1122.A_0082_EPP2817_0008_0017.DIG_Inputs_Device.Safe_state_active <-> DIG Inputs Device/Safe state active
//     PlcTask Inputs/GVL_iXlinker.EtherCAT_Master_EPPxxxx.Beckhoff_EPP2xxx.Beckhoff_EPP2xxxEK1122.A_0082_EPP2817_0008_0017.DIG_Inputs_Device.Error_channel[0] <-> DIG Inputs Device/Error channel 1
//     PlcTask Inputs/GVL_iXlinker.EtherCAT_Master_EPPxxxx.Beckhoff_EPP2xxx.Beckhoff_EPP2xxxEK1122.A_0082_EPP2817_0008_0017.DIG_Inputs_Device.Error_channel[1] <-> DIG Inputs Device/Error channel 2
//     PlcTask Inputs/GVL_iXlinker.EtherCAT_Master_EPPxxxx.Beckhoff_EPP2xxx.Beckhoff_EPP2xxxEK1122.A_0082_EPP2817_0008_0017.DIG_Inputs_Device.Error_channel[2] <-> DIG Inputs Device/Error channel 3
//     PlcTask Inputs/GVL_iXlinker.EtherCAT_Master_EPPxxxx.Beckhoff_EPP2xxx.Beckhoff_EPP2xxxEK1122.A_0082_EPP2817_0008_0017.DIG_Inputs_Device.Us_Undervoltage <-> DIG Inputs Device/Us Undervoltage
//     PlcTask Inputs/GVL_iXlinker.EtherCAT_Master_EPPxxxx.Beckhoff_EPP2xxx.Beckhoff_EPP2xxxEK1122.A_0082_EPP2817_0008_0017.DIG_Inputs_Device.Up_Undervoltage <-> DIG Inputs Device/Up Undervoltage
//     PlcTask Inputs/GVL_iXlinker.EtherCAT_Master_EPPxxxx.Beckhoff_EPP2xxx.Beckhoff_EPP2xxxEK1122.A_0082_EPP2817_0008_0017.DIG_Inputs_Device.Sync_error <-> DIG Inputs Device/Sync error
//     PlcTask Inputs/GVL_iXlinker.EtherCAT_Master_EPPxxxx.Beckhoff_EPP2xxx.Beckhoff_EPP2xxxEK1122.A_0082_EPP2817_0008_0017.DIG_Inputs_Device.TxPDO_Toggle <-> DIG Inputs Device/TxPDO Toggle
//     PlcTask Outputs/GVL_iXlinker.EtherCAT_Master_EPPxxxx.Beckhoff_EPP2xxx.Beckhoff_EPP2xxxEK1122.A_0082_EPP2817_0008_0017.DIG_Output_Channel_1.Output[0] <-> DIG Output Channel 1/Output 1
//     PlcTask Outputs/GVL_iXlinker.EtherCAT_Master_EPPxxxx.Beckhoff_EPP2xxx.Beckhoff_EPP2xxxEK1122.A_0082_EPP2817_0008_0017.DIG_Output_Channel_1.Output[1] <-> DIG Output Channel 1/Output 2
//     PlcTask Outputs/GVL_iXlinker.EtherCAT_Master_EPPxxxx.Beckhoff_EPP2xxx.Beckhoff_EPP2xxxEK1122.A_0082_EPP2817_0008_0017.DIG_Output_Channel_1.Output[2] <-> DIG Output Channel 1/Output 3
//     PlcTask Outputs/GVL_iXlinker.EtherCAT_Master_EPPxxxx.Beckhoff_EPP2xxx.Beckhoff_EPP2xxxEK1122.A_0082_EPP2817_0008_0017.DIG_Output_Channel_1.Output[3] <-> DIG Output Channel 1/Output 4
//     PlcTask Outputs/GVL_iXlinker.EtherCAT_Master_EPPxxxx.Beckhoff_EPP2xxx.Beckhoff_EPP2xxxEK1122.A_0082_EPP2817_0008_0017.DIG_Output_Channel_1.Output[4] <-> DIG Output Channel 1/Output 5
//     PlcTask Outputs/GVL_iXlinker.EtherCAT_Master_EPPxxxx.Beckhoff_EPP2xxx.Beckhoff_EPP2xxxEK1122.A_0082_EPP2817_0008_0017.DIG_Output_Channel_1.Output[5] <-> DIG Output Channel 1/Output 6
//     PlcTask Outputs/GVL_iXlinker.EtherCAT_Master_EPPxxxx.Beckhoff_EPP2xxx.Beckhoff_EPP2xxxEK1122.A_0082_EPP2817_0008_0017.DIG_Output_Channel_1.Output[6] <-> DIG Output Channel 1/Output 7
//     PlcTask Outputs/GVL_iXlinker.EtherCAT_Master_EPPxxxx.Beckhoff_EPP2xxx.Beckhoff_EPP2xxxEK1122.A_0082_EPP2817_0008_0017.DIG_Output_Channel_1.Output[7] <-> DIG Output Channel 1/Output 8
//     PlcTask Outputs/GVL_iXlinker.EtherCAT_Master_EPPxxxx.Beckhoff_EPP2xxx.Beckhoff_EPP2xxxEK1122.A_0082_EPP2817_0008_0017.DIG_Output_Channel_2.Output[0] <-> DIG Output Channel 2/Output 1
//     PlcTask Outputs/GVL_iXlinker.EtherCAT_Master_EPPxxxx.Beckhoff_EPP2xxx.Beckhoff_EPP2xxxEK1122.A_0082_EPP2817_0008_0017.DIG_Output_Channel_2.Output[1] <-> DIG Output Channel 2/Output 2
//     PlcTask Outputs/GVL_iXlinker.EtherCAT_Master_EPPxxxx.Beckhoff_EPP2xxx.Beckhoff_EPP2xxxEK1122.A_0082_EPP2817_0008_0017.DIG_Output_Channel_2.Output[2] <-> DIG Output Channel 2/Output 3
//     PlcTask Outputs/GVL_iXlinker.EtherCAT_Master_EPPxxxx.Beckhoff_EPP2xxx.Beckhoff_EPP2xxxEK1122.A_0082_EPP2817_0008_0017.DIG_Output_Channel_2.Output[3] <-> DIG Output Channel 2/Output 4
//     PlcTask Outputs/GVL_iXlinker.EtherCAT_Master_EPPxxxx.Beckhoff_EPP2xxx.Beckhoff_EPP2xxxEK1122.A_0082_EPP2817_0008_0017.DIG_Output_Channel_2.Output[4] <-> DIG Output Channel 2/Output 5
//     PlcTask Outputs/GVL_iXlinker.EtherCAT_Master_EPPxxxx.Beckhoff_EPP2xxx.Beckhoff_EPP2xxxEK1122.A_0082_EPP2817_0008_0017.DIG_Output_Channel_2.Output[5] <-> DIG Output Channel 2/Output 6
//     PlcTask Outputs/GVL_iXlinker.EtherCAT_Master_EPPxxxx.Beckhoff_EPP2xxx.Beckhoff_EPP2xxxEK1122.A_0082_EPP2817_0008_0017.DIG_Output_Channel_2.Output[6] <-> DIG Output Channel 2/Output 7
//     PlcTask Outputs/GVL_iXlinker.EtherCAT_Master_EPPxxxx.Beckhoff_EPP2xxx.Beckhoff_EPP2xxxEK1122.A_0082_EPP2817_0008_0017.DIG_Output_Channel_2.Output[7] <-> DIG Output Channel 2/Output 8
//     PlcTask Outputs/GVL_iXlinker.EtherCAT_Master_EPPxxxx.Beckhoff_EPP2xxx.Beckhoff_EPP2xxxEK1122.A_0082_EPP2817_0008_0017.DIG_Output_Channel_3.Output[0] <-> DIG Output Channel 3/Output 1
//     PlcTask Outputs/GVL_iXlinker.EtherCAT_Master_EPPxxxx.Beckhoff_EPP2xxx.Beckhoff_EPP2xxxEK1122.A_0082_EPP2817_0008_0017.DIG_Output_Channel_3.Output[1] <-> DIG Output Channel 3/Output 2
//     PlcTask Outputs/GVL_iXlinker.EtherCAT_Master_EPPxxxx.Beckhoff_EPP2xxx.Beckhoff_EPP2xxxEK1122.A_0082_EPP2817_0008_0017.DIG_Output_Channel_3.Output[2] <-> DIG Output Channel 3/Output 3
//     PlcTask Outputs/GVL_iXlinker.EtherCAT_Master_EPPxxxx.Beckhoff_EPP2xxx.Beckhoff_EPP2xxxEK1122.A_0082_EPP2817_0008_0017.DIG_Output_Channel_3.Output[3] <-> DIG Output Channel 3/Output 4
//     PlcTask Outputs/GVL_iXlinker.EtherCAT_Master_EPPxxxx.Beckhoff_EPP2xxx.Beckhoff_EPP2xxxEK1122.A_0082_EPP2817_0008_0017.DIG_Output_Channel_3.Output[4] <-> DIG Output Channel 3/Output 5
//     PlcTask Outputs/GVL_iXlinker.EtherCAT_Master_EPPxxxx.Beckhoff_EPP2xxx.Beckhoff_EPP2xxxEK1122.A_0082_EPP2817_0008_0017.DIG_Output_Channel_3.Output[5] <-> DIG Output Channel 3/Output 6
//     PlcTask Outputs/GVL_iXlinker.EtherCAT_Master_EPPxxxx.Beckhoff_EPP2xxx.Beckhoff_EPP2xxxEK1122.A_0082_EPP2817_0008_0017.DIG_Output_Channel_3.Output[6] <-> DIG Output Channel 3/Output 7
//     PlcTask Outputs/GVL_iXlinker.EtherCAT_Master_EPPxxxx.Beckhoff_EPP2xxx.Beckhoff_EPP2xxxEK1122.A_0082_EPP2817_0008_0017.DIG_Output_Channel_3.Output[7] <-> DIG Output Channel 3/Output 8
//     PlcTask Outputs/GVL_iXlinker.EtherCAT_Master_EPPxxxx.Beckhoff_EPP2xxx.Beckhoff_EPP2xxxEK1122.A_0082_EPP2817_0008_0017.DIG_Outputs_Device.Set_safe_state <-> DIG Outputs Device/Set safe state
//     PlcTask Outputs/GVL_iXlinker.EtherCAT_Master_EPPxxxx.Beckhoff_EPP2xxx.Beckhoff_EPP2xxxEK1122.A_0082_EPP2817_0008_0017.DIG_Outputs_Device.Reset_outputs <-> DIG Outputs Device/Reset outputs
//     PlcTask Inputs/GVL_iXlinker.EtherCAT_Master_EPPxxxx.Beckhoff_EPP2xxx.Beckhoff_EPP2xxxEK1122.A_0082_EPP2817_0008_0017.WcState.WcState <-> WcState/WcState
//     PlcTask Inputs/GVL_iXlinker.EtherCAT_Master_EPPxxxx.Beckhoff_EPP2xxx.Beckhoff_EPP2xxxEK1122.A_0082_EPP2817_0008_0017.WcState.InputToggle <-> WcState/InputToggle
//     PlcTask Inputs/GVL_iXlinker.EtherCAT_Master_EPPxxxx.Beckhoff_EPP2xxx.Beckhoff_EPP2xxxEK1122.A_0082_EPP2817_0008_0017.InfoData.AdsAddr <-> InfoData/AdsAddr
//     PlcTask Inputs/GVL_iXlinker.EtherCAT_Master_EPPxxxx.Beckhoff_EPP2xxx.Beckhoff_EPP2xxxEK1122.A_0082_EPP2817_0008_0017.InfoData.State <-> InfoData/State
//   PLC/PLC Instance <-> EtherCAT Master EPPxxxx/Beckhoff EPP2xxx/Beckhoff EPP2xxxEK1122/A_0083(EPP2817-0008-0018)
//     PlcTask Inputs/GVL_iXlinker.EtherCAT_Master_EPPxxxx.Beckhoff_EPP2xxx.Beckhoff_EPP2xxxEK1122.A_0083_EPP2817_0008_0018.DIG_Diag_Inputs_Channel_1.Diag_Input[0] <-> DIG Diag Inputs Channel 1/Diag Input 1
//     PlcTask Inputs/GVL_iXlinker.EtherCAT_Master_EPPxxxx.Beckhoff_EPP2xxx.Beckhoff_EPP2xxxEK1122.A_0083_EPP2817_0008_0018.DIG_Diag_Inputs_Channel_1.Diag_Input[1] <-> DIG Diag Inputs Channel 1/Diag Input 2
//     PlcTask Inputs/GVL_iXlinker.EtherCAT_Master_EPPxxxx.Beckhoff_EPP2xxx.Beckhoff_EPP2xxxEK1122.A_0083_EPP2817_0008_0018.DIG_Diag_Inputs_Channel_1.Diag_Input[2] <-> DIG Diag Inputs Channel 1/Diag Input 3
//     PlcTask Inputs/GVL_iXlinker.EtherCAT_Master_EPPxxxx.Beckhoff_EPP2xxx.Beckhoff_EPP2xxxEK1122.A_0083_EPP2817_0008_0018.DIG_Diag_Inputs_Channel_1.Diag_Input[3] <-> DIG Diag Inputs Channel 1/Diag Input 4
//     PlcTask Inputs/GVL_iXlinker.EtherCAT_Master_EPPxxxx.Beckhoff_EPP2xxx.Beckhoff_EPP2xxxEK1122.A_0083_EPP2817_0008_0018.DIG_Diag_Inputs_Channel_1.Diag_Input[4] <-> DIG Diag Inputs Channel 1/Diag Input 5
//     PlcTask Inputs/GVL_iXlinker.EtherCAT_Master_EPPxxxx.Beckhoff_EPP2xxx.Beckhoff_EPP2xxxEK1122.A_0083_EPP2817_0008_0018.DIG_Diag_Inputs_Channel_1.Diag_Input[5] <-> DIG Diag Inputs Channel 1/Diag Input 6
//     PlcTask Inputs/GVL_iXlinker.EtherCAT_Master_EPPxxxx.Beckhoff_EPP2xxx.Beckhoff_EPP2xxxEK1122.A_0083_EPP2817_0008_0018.DIG_Diag_Inputs_Channel_1.Diag_Input[6] <-> DIG Diag Inputs Channel 1/Diag Input 7
//     PlcTask Inputs/GVL_iXlinker.EtherCAT_Master_EPPxxxx.Beckhoff_EPP2xxx.Beckhoff_EPP2xxxEK1122.A_0083_EPP2817_0008_0018.DIG_Diag_Inputs_Channel_1.Diag_Input[7] <-> DIG Diag Inputs Channel 1/Diag Input 8
//     PlcTask Inputs/GVL_iXlinker.EtherCAT_Master_EPPxxxx.Beckhoff_EPP2xxx.Beckhoff_EPP2xxxEK1122.A_0083_EPP2817_0008_0018.DIG_Diag_Inputs_Channel_2.Diag_Input[0] <-> DIG Diag Inputs Channel 2/Diag Input 1
